LIN {X 0,Y 369.377,Z 414.803,A -85,B 0,C 180,E1 -12869.73,E2 -12869.73} C_VEL
LIN {X 0,Y 368.676,Z 422.155,A -85,B 0,C 180,E1 -12871.367,E2 -12871.367} C_VEL
LIN {X 0,Y 368.229,Z 428.905,A -85,B 0,C 180,E1 -12873.284,E2 -12873.284} C_VEL
LIN {X 0,Y 367.894,Z 433.372,A -85,B 0,C 180,E1 -12874.933,E2 -12874.933} C_VEL
LIN {X 0,Y 367.73,Z 436.765,A -85,B 0,C 180,E1 -12876.586,E2 -12876.586} C_VEL
LIN {X 0,Y 367.581,Z 438.459,A -85,B 0,C 180,E1 -12877.693,E2 -12877.693} C_VEL
LIN {X 0,Y 367.47,Z 439.751,A -85,B 0,C 180,E1 -12878.802,E2 -12878.802} C_VEL
LIN {X 0,Y 367.38,Z 440.649,A -85,B 0,C 180,E1 -12879.915,E2 -12879.915} C_VEL
LIN {X 0,Y 367.424,Z 441.1,A -85,B 0,C 180,E1 -12881.028,E2 -12881.028} C_VEL
LIN {X 0,Y 367.521,Z 441.023,A -85,B 0,C 180,E1 -12882.77,E2 -12882.77} C_VEL
LIN {X 0,Y 367.587,Z 440.078,A -85,B 0,C 180,E1 -12884.392,E2 -12884.392} C_VEL
LIN {X 0,Y 367.854,Z 438.002,A -85,B 0,C 180,E1 -12886.13,E2 -12886.13} C_VEL
LIN {X 0,Y 368.254,Z 435.208,A -85,B 0,C 180,E1 -12887.78,E2 -12887.78} C_VEL
LIN {X 0,Y 368.738,Z 431.176,A -85,B 0,C 180,E1 -12889.484,E2 -12889.484} C_VEL
LIN {X 0,Y 369.195,Z 427.833,A -85,B 0,C 180,E1 -12890.605,E2 -12890.605} C_VEL
LIN {X 0,Y 368.924,Z 425.231,A -85,B 0,C 180,E1 -12891.428,E2 -12891.428} C_VEL
LIN {X 0,Y 366.799,Z 420.655,A -85,B 0,C 180,E1 -12892.758,E2 -12892.758} C_VEL
LIN {X 0,Y 364.754,Z 415.467,A -85,B 0,C 180,E1 -12894.041,E2 -12894.041} C_VEL
LIN {X 0,Y 364.604,Z 411.868,A -85,B 0,C 180,E1 -12894.779,E2 -12894.779} C_VEL
LIN {X 0,Y 365.717,Z 403.299,A -85,B 0,C 180,E1 -12896.231,E2 -12896.231} C_VEL
LIN {X 0,Y 366.895,Z 393.904,A -85,B 0,C 180,E1 -12897.523,E2 -12897.523} C_VEL
LIN {X 0,Y 368.133,Z 383.723,A -85,B 0,C 180,E1 -12898.647,E2 -12898.647} C_VEL
LIN {X 0,Y 369.203,Z 372.197,A -85,B 0,C 180,E1 -12899.664,E2 -12899.664} C_VEL
LIN {X 0,Y 370.055,Z 360.622,A -85,B 0,C 180,E1 -12900.453,E2 -12900.453} C_VEL
LIN {X 0,Y 370.819,Z 347.971,A -85,B 0,C 180,E1 -12901.072,E2 -12901.072} C_VEL
LIN {X 0,Y 371.327,Z 334.426,A -85,B 0,C 180,E1 -12901.491,E2 -12901.491} C_VEL
LIN {X 0,Y 372.84,Z 255.873,A -85,B 0,C 180,E1 -12903.038,E2 -12903.038} C_VEL
LIN {X 0,Y 370.773,Z 248.12,A -85,B 0,C 180,E1 -12903.357,E2 -12903.357} C_VEL
LIN {X 0,Y 363.463,Z 231.06,A -85,B 0,C 180,E1 -12904.307,E2 -12904.307} C_VEL
LIN {X 0,Y 361.887,Z 224.41,A -85,B 0,C 180,E1 -12906.234,E2 -12906.234} C_VEL
LIN {X 0,Y 361.876,Z 224.407,A -85,B 0,C 180,E1 -12909.857,E2 -12909.857} C_VEL
LIN {X 0,Y 361.848,Z 224.414,A -85,B 0,C 180,E1 -12912.825,E2 -12912.825} C_VEL
LIN {X 0,Y 361.888,Z 224.41,A -85,B 0,C 180,E1 -12915.932,E2 -12915.932} C_VEL
LIN {X 0,Y 361.896,Z 224.406,A -85,B 0,C 180,E1 -12919.23,E2 -12919.23} C_VEL
LIN {X 0,Y 361.856,Z 224.406,A -85,B 0,C 180,E1 -12922.98,E2 -12922.98} C_VEL
LIN {X 0,Y 361.845,Z 224.411,A -85,B 0,C 180,E1 -12926.629,E2 -12926.629} C_VEL
LIN {X 0,Y 361.861,Z 224.406,A -85,B 0,C 180,E1 -12929.67,E2 -12929.67} C_VEL
LIN {X 0,Y 361.937,Z 224.396,A -85,B 0,C 180,E1 -12933.473,E2 -12933.473} C_VEL
LIN {X 0,Y 361.859,Z 224.404,A -85,B 0,C 180,E1 -12937.142,E2 -12937.142} C_VEL
LIN {X 0,Y 361.862,Z 224.401,A -85,B 0,C 180,E1 -12940.721,E2 -12940.721} C_VEL
LIN {X 0,Y 361.912,Z 224.403,A -85,B 0,C 180,E1 -12943.065,E2 -12943.065} C_VEL
LIN {X 0,Y 361.976,Z 224.393,A -85,B 0,C 180,E1 -12946.527,E2 -12946.527} C_VEL
LIN {X 0,Y 362.007,Z 224.39,A -85,B 0,C 180,E1 -12949.937,E2 -12949.937} C_VEL
LIN {X 0,Y 362.141,Z 224.37,A -85,B 0,C 180,E1 -12953.313,E2 -12953.313} C_VEL
LIN {X 0,Y 362.252,Z 224.352,A -85,B 0,C 180,E1 -12957.776,E2 -12957.776} C_VEL
LIN {X 0,Y 362.379,Z 224.343,A -85,B 0,C 180,E1 -12960,E2 -12960} C_VEL
LIN {X 0,Y 362.252,Z 224.355,A -85,B 0,C 180,E1 -12962.224,E2 -12962.224} C_VEL
LIN {X 0,Y 362.113,Z 224.377,A -85,B 0,C 180,E1 -12966.687,E2 -12966.687} C_VEL
LIN {X 0,Y 361.977,Z 224.393,A -85,B 0,C 180,E1 -12970.063,E2 -12970.063} C_VEL
LIN {X 0,Y 361.977,Z 224.392,A -85,B 0,C 180,E1 -12973.899,E2 -12973.899} C_VEL
LIN {X 0,Y 361.907,Z 224.398,A -85,B 0,C 180,E1 -12976.935,E2 -12976.935} C_VEL
LIN {X 0,Y 361.854,Z 224.409,A -85,B 0,C 180,E1 -12980.463,E2 -12980.463} C_VEL
LIN {X 0,Y 361.843,Z 224.411,A -85,B 0,C 180,E1 -12984.102,E2 -12984.102} C_VEL
LIN {X 0,Y 361.826,Z 224.413,A -85,B 0,C 180,E1 -12987.786,E2 -12987.786} C_VEL
LIN {X 0,Y 361.81,Z 224.415,A -85,B 0,C 180,E1 -12991.281,E2 -12991.281} C_VEL
LIN {X 0,Y 361.835,Z 224.408,A -85,B 0,C 180,E1 -12994.283,E2 -12994.283} C_VEL
LIN {X 0,Y 361.845,Z 224.4,A -85,B 0,C 180,E1 -12997.223,E2 -12997.223} C_VEL
LIN {X 0,Y 361.822,Z 224.415,A -85,B 0,C 180,E1 -13000.756,E2 -13000.756} C_VEL
LIN {X 0,Y 361.806,Z 224.418,A -85,B 0,C 180,E1 -13004.37,E2 -13004.37} C_VEL
LIN {X 0,Y 361.822,Z 224.41,A -85,B 0,C 180,E1 -13007.571,E2 -13007.571} C_VEL
LIN {X 0,Y 361.836,Z 224.407,A -85,B 0,C 180,E1 -13011.573,E2 -13011.573} C_VEL
LIN {X 0,Y 361.87,Z 224.404,A -85,B 0,C 180,E1 -13014.656,E2 -13014.656} C_VEL
LIN {X 0,Y 361.907,Z 224.589,A -85,B 0,C 180,E1 -13018.051,E2 -13018.051} C_VEL
LIN {X 0,Y 365.046,Z 237.635,A -85,B 0,C 180,E1 -13021.507,E2 -13021.507} C_VEL
LIN {X 0,Y 366.873,Z 247.039,A -85,B 0,C 180,E1 -13023.858,E2 -13023.858} C_VEL
LIN {X 0,Y 366,Z 256.31,A -85,B 0,C 180,E1 -13025.918,E2 -13025.918} C_VEL
LIN {X 0,Y 365.489,Z 261.029,A -85,B 0,C 180,E1 -13026.928,E2 -13026.928} C_VEL
LIN {X 0,Y 370.101,Z 284.638,A -85,B 0,C 180,E1 -13027.78,E2 -13027.78} C_VEL
LIN {X 0,Y 372.121,Z 298.577,A -85,B 0,C 180,E1 -13028.219,E2 -13028.219} C_VEL
LIN {X 0,Y 370.713,Z 370.18,A -85,B 0,C 180,E1 -13029.649,E2 -13029.649} C_VEL
LIN {X 0,Y 369.936,Z 383.988,A -85,B 0,C 180,E1 -13030.148,E2 -13030.148} C_VEL
LIN {X 0,Y 368.872,Z 396.399,A -85,B 0,C 180,E1 -13030.812,E2 -13030.812} C_VEL
LIN {X 0,Y 367.758,Z 407.492,A -85,B 0,C 180,E1 -13031.619,E2 -13031.619} C_VEL
LIN {X 0,Y 366.392,Z 419.049,A -85,B 0,C 180,E1 -13032.703,E2 -13032.703} C_VEL
LIN {X 0,Y 365.116,Z 429.47,A -85,B 0,C 180,E1 -13033.936,E2 -13033.936} C_VEL
LIN {X 0,Y 363.969,Z 438.334,A -85,B 0,C 180,E1 -13035.227,E2 -13035.227} C_VEL
LIN {X 0,Y 362.841,Z 447.307,A -85,B 0,C 180,E1 -13036.844,E2 -13036.844} C_VEL
LIN {X 0,Y 361.793,Z 454.782,A -85,B 0,C 180,E1 -13038.514,E2 -13038.514} C_VEL
LIN {X 0,Y 361.043,Z 461.718,A -85,B 0,C 180,E1 -13040.475,E2 -13040.475} C_VEL
LIN {X 0,Y 360.649,Z 466.318,A -85,B 0,C 180,E1 -13042.159,E2 -13042.159} C_VEL
LIN {X 0,Y 360.424,Z 470.058,A -85,B 0,C 180,E1 -13043.969,E2 -13043.969} C_VEL
LIN {X 0,Y 360.364,Z 472.357,A -85,B 0,C 180,E1 -13045.524,E2 -13045.524} C_VEL
LIN {X 0,Y 360.321,Z 473.53,A -85,B 0,C 180,E1 -13046.644,E2 -13046.644} C_VEL
LIN {X 0,Y 360.454,Z 474.635,A -85,B 0,C 180,E1 -13048.881,E2 -13048.881} C_VEL
LIN {X 0,Y 360.48,Z 474.606,A -85,B 0,C 180,E1 -13049.998,E2 -13049.998} C_VEL
LIN {X 0,Y 360.476,Z 474.176,A -85,B 0,C 180,E1 -13051.115,E2 -13051.115} C_VEL
LIN {X 0,Y 360.395,Z 473.302,A -85,B 0,C 180,E1 -13052.233,E2 -13052.233} C_VEL
LIN {X 0,Y 360.436,Z 470.349,A -85,B 0,C 180,E1 -13054.471,E2 -13054.471} C_VEL
LIN {X 0,Y 360.442,Z 467.158,A -85,B 0,C 180,E1 -13056.059,E2 -13056.059} C_VEL
LIN {X 0,Y 360.637,Z 462.452,A -85,B 0,C 180,E1 -13057.837,E2 -13057.837} C_VEL
LIN {X 0,Y 361.013,Z 455.625,A -85,B 0,C 180,E1 -13059.804,E2 -13059.804} C_VEL
LIN {X 0,Y 361.56,Z 448.175,A -85,B 0,C 180,E1 -13061.489,E2 -13061.489} C_VEL
LIN {X 0,Y 362.248,Z 440.586,A -85,B 0,C 180,E1 -13062.888,E2 -13062.888} C_VEL
LIN {X 0,Y 363.021,Z 432.028,A -85,B 0,C 180,E1 -13064.194,E2 -13064.194} C_VEL
LIN {X 0,Y 363.918,Z 421.306,A -85,B 0,C 180,E1 -13065.524,E2 -13065.524} C_VEL
LIN {X 0,Y 364.862,Z 409.823,A -85,B 0,C 180,E1 -13066.646,E2 -13066.646} C_VEL
LIN {X 0,Y 365.769,Z 398.067,A -85,B 0,C 180,E1 -13067.539,E2 -13067.539} C_VEL
LIN {X 0,Y 366.614,Z 385.299,A -85,B 0,C 180,E1 -13068.255,E2 -13068.255} C_VEL
LIN {X 0,Y 367.305,Z 371.702,A -85,B 0,C 180,E1 -13068.761,E2 -13068.761} C_VEL
LIN {X 0,Y 367.865,Z 337.148,A -85,B 0,C 180,E1 -13069.469,E2 -13069.469} C_VEL
LIN {X 0,Y 368.221,Z 295.328,A -85,B 0,C 180,E1 -13070.291,E2 -13070.291} C_VEL
LIN {X 0,Y 363.689,Z 261.477,A -85,B 0,C 180,E1 -13071.21,E2 -13071.21} C_VEL
LIN {X 0,Y 365.131,Z 243.552,A -85,B 0,C 180,E1 -13075.048,E2 -13075.048} C_VEL
LIN {X 0,Y 364.937,Z 239.311,A -85,B 0,C 180,E1 -13075.993,E2 -13075.993} C_VEL
LIN {X 0,Y 362.387,Z 226.582,A -85,B 0,C 180,E1 -13078.997,E2 -13078.997} C_VEL
LIN {X 0,Y 361.891,Z 224.407,A -85,B 0,C 180,E1 -13079.546,E2 -13079.546} C_VEL
LIN {X 0,Y 361.841,Z 224.41,A -85,B 0,C 180,E1 -13083.365,E2 -13083.365} C_VEL
LIN {X 0,Y 361.846,Z 224.408,A -85,B 0,C 180,E1 -13087.014,E2 -13087.014} C_VEL
LIN {X 0,Y 361.831,Z 224.416,A -85,B 0,C 180,E1 -13089.857,E2 -13089.857} C_VEL
LIN {X 0,Y 361.812,Z 224.413,A -85,B 0,C 180,E1 -13092.824,E2 -13092.824} C_VEL
LIN {X 0,Y 361.868,Z 224.411,A -85,B 0,C 180,E1 -13095.93,E2 -13095.93} C_VEL
LIN {X 0,Y 361.876,Z 224.406,A -85,B 0,C 180,E1 -13099.228,E2 -13099.228} C_VEL
LIN {X 0,Y 361.834,Z 224.41,A -85,B 0,C 180,E1 -13102.978,E2 -13102.978} C_VEL
LIN {X 0,Y 361.822,Z 224.411,A -85,B 0,C 180,E1 -13106.627,E2 -13106.627} C_VEL
LIN {X 0,Y 361.837,Z 224.415,A -85,B 0,C 180,E1 -13109.669,E2 -13109.669} C_VEL
LIN {X 0,Y 361.913,Z 224.406,A -85,B 0,C 180,E1 -13113.472,E2 -13113.472} C_VEL
LIN {X 0,Y 361.879,Z 224.407,A -85,B 0,C 180,E1 -13117.144,E2 -13117.144} C_VEL
LIN {X 0,Y 361.89,Z 224.404,A -85,B 0,C 180,E1 -13120.722,E2 -13120.722} C_VEL
LIN {X 0,Y 361.9,Z 224.402,A -85,B 0,C 180,E1 -13124.224,E2 -13124.224} C_VEL
LIN {X 0,Y 361.952,Z 224.395,A -85,B 0,C 180,E1 -13126.526,E2 -13126.526} C_VEL
LIN {X 0,Y 361.988,Z 224.391,A -85,B 0,C 180,E1 -13129.937,E2 -13129.937} C_VEL
LIN {X 0,Y 362.101,Z 224.377,A -85,B 0,C 180,E1 -13132.192,E2 -13132.192} C_VEL
LIN {X 0,Y 362.075,Z 224.38,A -85,B 0,C 180,E1 -13134.431,E2 -13134.431} C_VEL
LIN {X 0,Y 362.232,Z 224.361,A -85,B 0,C 180,E1 -13137.776,E2 -13137.776} C_VEL
LIN {X 0,Y 362.376,Z 224.342,A -85,B 0,C 180,E1 -13140,E2 -13140} C_VEL
LIN {X 0,Y 362.228,Z 224.361,A -85,B 0,C 180,E1 -13142.224,E2 -13142.224} C_VEL
LIN {X 0,Y 362.111,Z 224.379,A -85,B 0,C 180,E1 -13146.687,E2 -13146.687} C_VEL
LIN {X 0,Y 361.985,Z 224.391,A -85,B 0,C 180,E1 -13150.063,E2 -13150.063} C_VEL
LIN {X 0,Y 361.952,Z 224.395,A -85,B 0,C 180,E1 -13153.9,E2 -13153.9} C_VEL
LIN {X 0,Y 361.908,Z 224.401,A -85,B 0,C 180,E1 -13157.933,E2 -13157.933} C_VEL
LIN {X 0,Y 361.817,Z 224.412,A -85,B 0,C 180,E1 -13161.658,E2 -13161.658} C_VEL
LIN {X 0,Y 361.884,Z 224.404,A -85,B 0,C 180,E1 -13165.294,E2 -13165.294} C_VEL
LIN {X 0,Y 361.879,Z 224.405,A -85,B 0,C 180,E1 -13167.782,E2 -13167.782} C_VEL
LIN {X 0,Y 361.81,Z 224.413,A -85,B 0,C 180,E1 -13171.289,E2 -13171.289} C_VEL
LIN {X 0,Y 361.818,Z 224.416,A -85,B 0,C 180,E1 -13174.285,E2 -13174.285} C_VEL
LIN {X 0,Y 361.83,Z 224.41,A -85,B 0,C 180,E1 -13177.227,E2 -13177.227} C_VEL
LIN {X 0,Y 361.877,Z 224.407,A -85,B 0,C 180,E1 -13180.773,E2 -13180.773} C_VEL
LIN {X 0,Y 361.874,Z 224.41,A -85,B 0,C 180,E1 -13184.36,E2 -13184.36} C_VEL
LIN {X 0,Y 361.812,Z 224.413,A -85,B 0,C 180,E1 -13187.573,E2 -13187.573} C_VEL
LIN {X 0,Y 361.848,Z 224.408,A -85,B 0,C 180,E1 -13190.978,E2 -13190.978} C_VEL
LIN {X 0,Y 361.856,Z 224.408,A -85,B 0,C 180,E1 -13194.66,E2 -13194.66} C_VEL
LIN {X 0,Y 361.823,Z 224.414,A -85,B 0,C 180,E1 -13198.375,E2 -13198.375} C_VEL
LIN {X 0,Y 361.896,Z 224.406,A -85,B 0,C 180,E1 -13202.225,E2 -13202.225} C_VEL
LIN {X 0,Y 361.917,Z 224.4,A -85,B 0,C 180,E1 -13204.714,E2 -13204.714} C_VEL
LIN {X 0,Y 361.854,Z 224.409,A -85,B 0,C 180,E1 -13208.349,E2 -13208.349} C_VEL
LIN {X 0,Y 361.916,Z 224.403,A -85,B 0,C 180,E1 -13212.088,E2 -13212.088} C_VEL
LIN {X 0,Y 361.959,Z 224.397,A -85,B 0,C 180,E1 -13215.383,E2 -13215.383} C_VEL
LIN {X 0,Y 362.005,Z 224.579,A -85,B 0,C 180,E1 -13218.312,E2 -13218.312} C_VEL
LIN {X 0,Y 363.238,Z 230.767,A -85,B 0,C 180,E1 -13219.872,E2 -13219.872} C_VEL
LIN {X 0,Y 366.475,Z 241.241,A -85,B 0,C 180,E1 -13220.25,E2 -13220.25} C_VEL
LIN {X 0,Y 368.895,Z 254.352,A -85,B 0,C 180,E1 -13220.635,E2 -13220.635} C_VEL
LIN {X 0,Y 367.507,Z 337.938,A -85,B 0,C 180,E1 -13222.275,E2 -13222.275} C_VEL
LIN {X 0,Y 367.022,Z 351.062,A -85,B 0,C 180,E1 -13222.749,E2 -13222.749} C_VEL
LIN {X 0,Y 366.477,Z 363.096,A -85,B 0,C 180,E1 -13223.395,E2 -13223.395} C_VEL
LIN {X 0,Y 365.943,Z 374.427,A -85,B 0,C 180,E1 -13224.216,E2 -13224.216} C_VEL
LIN {X 0,Y 364.895,Z 386.165,A -85,B 0,C 180,E1 -13225.307,E2 -13225.307} C_VEL
LIN {X 0,Y 364.001,Z 396.644,A -85,B 0,C 180,E1 -13226.543,E2 -13226.543} C_VEL
LIN {X 0,Y 363.227,Z 405.215,A -85,B 0,C 180,E1 -13227.785,E2 -13227.785} C_VEL
LIN {X 0,Y 362.557,Z 413.108,A -85,B 0,C 180,E1 -13229.169,E2 -13229.169} C_VEL
LIN {X 0,Y 361.754,Z 420.868,A -85,B 0,C 180,E1 -13230.837,E2 -13230.837} C_VEL
LIN {X 0,Y 361.263,Z 427.957,A -85,B 0,C 180,E1 -13232.789,E2 -13232.789} C_VEL
LIN {X 0,Y 360.853,Z 432.71,A -85,B 0,C 180,E1 -13234.47,E2 -13234.47} C_VEL
LIN {X 0,Y 360.675,Z 436.807,A -85,B 0,C 180,E1 -13236.396,E2 -13236.396} C_VEL
LIN {X 0,Y 360.469,Z 438.987,A -85,B 0,C 180,E1 -13237.845,E2 -13237.845} C_VEL
LIN {X 0,Y 360.38,Z 440.234,A -85,B 0,C 180,E1 -13238.977,E2 -13238.977} C_VEL
LIN {X 0,Y 360.286,Z 441.057,A -85,B 0,C 180,E1 -13240.112,E2 -13240.112} C_VEL
LIN {X 0,Y 360.358,Z 441.451,A -85,B 0,C 180,E1 -13241.247,E2 -13241.247} C_VEL
LIN {X 0,Y 360.451,Z 441.352,A -85,B 0,C 180,E1 -13242.865,E2 -13242.865} C_VEL
LIN {X 0,Y 360.539,Z 440.257,A -85,B 0,C 180,E1 -13244.68,E2 -13244.68} C_VEL
LIN {X 0,Y 360.713,Z 439.007,A -85,B 0,C 180,E1 -13245.83,E2 -13245.83} C_VEL
LIN {X 0,Y 361.123,Z 436.391,A -85,B 0,C 180,E1 -13247.519,E2 -13247.519} C_VEL
LIN {X 0,Y 361.609,Z 432.561,A -85,B 0,C 180,E1 -13249.293,E2 -13249.293} C_VEL
LIN {X 0,Y 362.309,Z 427.786,A -85,B 0,C 180,E1 -13250.974,E2 -13250.974} C_VEL
LIN {X 0,Y 363.2,Z 421.309,A -85,B 0,C 180,E1 -13252.768,E2 -13252.768} C_VEL
LIN {X 0,Y 364.407,Z 413.357,A -85,B 0,C 180,E1 -13254.497,E2 -13254.497} C_VEL
LIN {X 0,Y 364.604,Z 411.868,A -85,B 0,C 180,E1 -13254.779,E2 -13254.779} C_VEL
LIN {X 0,Y 364.459,Z 408.101,A -85,B 0,C 180,E1 -13255.497,E2 -13255.497} C_VEL
LIN {X 0,Y 362.508,Z 401.791,A -85,B 0,C 180,E1 -13256.667,E2 -13256.667} C_VEL
LIN {X 0,Y 360.686,Z 395.024,A -85,B 0,C 180,E1 -13257.77,E2 -13257.77} C_VEL
LIN {X 0,Y 360.713,Z 390.444,A -85,B 0,C 180,E1 -13258.363,E2 -13258.363} C_VEL
LIN {X 0,Y 362.021,Z 379.271,A -85,B 0,C 180,E1 -13259.512,E2 -13259.512} C_VEL
LIN {X 0,Y 363.107,Z 366.471,A -85,B 0,C 180,E1 -13260.535,E2 -13260.535} C_VEL
LIN {X 0,Y 364.007,Z 354.12,A -85,B 0,C 180,E1 -13261.256,E2 -13261.256} C_VEL
LIN {X 0,Y 364.648,Z 340.948,A -85,B 0,C 180,E1 -13261.777,E2 -13261.777} C_VEL
LIN {X 0,Y 365.172,Z 319.833,A -85,B 0,C 180,E1 -13262.245,E2 -13262.245} C_VEL
LIN {X 0,Y 366.417,Z 257.084,A -85,B 0,C 180,E1 -13263.497,E2 -13263.497} C_VEL
LIN {X 0,Y 364.527,Z 250.334,A -85,B 0,C 180,E1 -13263.791,E2 -13263.791} C_VEL
LIN {X 0,Y 356.336,Z 231.44,A -85,B 0,C 180,E1 -13264.886,E2 -13264.886} C_VEL
LIN {X 0,Y 354.841,Z 225.287,A -85,B 0,C 180,E1 -13266.718,E2 -13266.718} C_VEL
LIN {X 0,Y 354.82,Z 225.289,A -85,B 0,C 180,E1 -13269.422,E2 -13269.422} C_VEL
LIN {X 0,Y 354.8,Z 225.292,A -85,B 0,C 180,E1 -13272.869,E2 -13272.869} C_VEL
LIN {X 0,Y 354.831,Z 225.291,A -85,B 0,C 180,E1 -13276.113,E2 -13276.113} C_VEL
LIN {X 0,Y 354.847,Z 225.284,A -85,B 0,C 180,E1 -13279.187,E2 -13279.187} C_VEL
LIN {X 0,Y 354.797,Z 225.286,A -85,B 0,C 180,E1 -13282.401,E2 -13282.401} C_VEL
LIN {X 0,Y 354.799,Z 225.287,A -85,B 0,C 180,E1 -13284.939,E2 -13284.939} C_VEL
LIN {X 0,Y 354.779,Z 225.287,A -85,B 0,C 180,E1 -13288.404,E2 -13288.404} C_VEL
LIN {X 0,Y 354.836,Z 225.284,A -85,B 0,C 180,E1 -13291.617,E2 -13291.617} C_VEL
LIN {X 0,Y 354.881,Z 225.28,A -85,B 0,C 180,E1 -13294.171,E2 -13294.171} C_VEL
LIN {X 0,Y 354.796,Z 225.292,A -85,B 0,C 180,E1 -13297.891,E2 -13297.891} C_VEL
LIN {X 0,Y 354.904,Z 225.278,A -85,B 0,C 180,E1 -13301.891,E2 -13301.891} C_VEL
LIN {X 0,Y 354.922,Z 225.274,A -85,B 0,C 180,E1 -13305.982,E2 -13305.982} C_VEL
LIN {X 0,Y 354.954,Z 225.267,A -85,B 0,C 180,E1 -13309.735,E2 -13309.735} C_VEL
LIN {X 0,Y 355.104,Z 225.247,A -85,B 0,C 180,E1 -13313.18,E2 -13313.18} C_VEL
LIN {X 0,Y 355.216,Z 225.229,A -85,B 0,C 180,E1 -13317.732,E2 -13317.732} C_VEL
LIN {X 0,Y 355.329,Z 225.221,A -85,B 0,C 180,E1 -13320,E2 -13320} C_VEL
LIN {X 0,Y 355.215,Z 225.232,A -85,B 0,C 180,E1 -13322.268,E2 -13322.268} C_VEL
LIN {X 0,Y 355.077,Z 225.251,A -85,B 0,C 180,E1 -13326.82,E2 -13326.82} C_VEL
LIN {X 0,Y 354.934,Z 225.27,A -85,B 0,C 180,E1 -13330.265,E2 -13330.265} C_VEL
LIN {X 0,Y 354.921,Z 225.271,A -85,B 0,C 180,E1 -13334.018,E2 -13334.018} C_VEL
LIN {X 0,Y 354.869,Z 225.275,A -85,B 0,C 180,E1 -13338.092,E2 -13338.092} C_VEL
LIN {X 0,Y 354.787,Z 225.283,A -85,B 0,C 180,E1 -13342.109,E2 -13342.109} C_VEL
LIN {X 0,Y 354.789,Z 225.281,A -85,B 0,C 180,E1 -13345.836,E2 -13345.836} C_VEL
LIN {X 0,Y 354.777,Z 225.285,A -85,B 0,C 180,E1 -13349.686,E2 -13349.686} C_VEL
LIN {X 0,Y 354.793,Z 225.282,A -85,B 0,C 180,E1 -13353.703,E2 -13353.703} C_VEL
LIN {X 0,Y 354.779,Z 225.286,A -85,B 0,C 180,E1 -13356.462,E2 -13356.462} C_VEL
LIN {X 0,Y 354.788,Z 225.275,A -85,B 0,C 180,E1 -13359.42,E2 -13359.42} C_VEL
LIN {X 0,Y 354.777,Z 225.29,A -85,B 0,C 180,E1 -13362.868,E2 -13362.868} C_VEL
LIN {X 0,Y 354.757,Z 225.296,A -85,B 0,C 180,E1 -13366.105,E2 -13366.105} C_VEL
LIN {X 0,Y 354.759,Z 225.29,A -85,B 0,C 180,E1 -13369.177,E2 -13369.177} C_VEL
LIN {X 0,Y 354.795,Z 225.286,A -85,B 0,C 180,E1 -13372.405,E2 -13372.405} C_VEL
LIN {X 0,Y 354.808,Z 225.284,A -85,B 0,C 180,E1 -13374.942,E2 -13374.942} C_VEL
LIN {X 0,Y 354.829,Z 225.45,A -85,B 0,C 180,E1 -13377.546,E2 -13377.546} C_VEL
LIN {X 0,Y 358.154,Z 239.13,A -85,B 0,C 180,E1 -13381.266,E2 -13381.266} C_VEL
LIN {X 0,Y 360.021,Z 248.666,A -85,B 0,C 180,E1 -13383.703,E2 -13383.703} C_VEL
LIN {X 0,Y 359.01,Z 258.823,A -85,B 0,C 180,E1 -13386.003,E2 -13386.003} C_VEL
LIN {X 0,Y 358.787,Z 260.543,A -85,B 0,C 180,E1 -13386.386,E2 -13386.386} C_VEL
LIN {X 0,Y 363.779,Z 286.169,A -85,B 0,C 180,E1 -13387.34,E2 -13387.34} C_VEL
LIN {X 0,Y 365.668,Z 298.645,A -85,B 0,C 180,E1 -13387.75,E2 -13387.75} C_VEL
LIN {X 0,Y 364.246,Z 369.797,A -85,B 0,C 180,E1 -13389.198,E2 -13389.198} C_VEL
LIN {X 0,Y 363.407,Z 383.627,A -85,B 0,C 180,E1 -13389.702,E2 -13389.702} C_VEL
LIN {X 0,Y 362.335,Z 396.043,A -85,B 0,C 180,E1 -13390.379,E2 -13390.379} C_VEL
LIN {X 0,Y 361.057,Z 407.925,A -85,B 0,C 180,E1 -13391.266,E2 -13391.266} C_VEL
LIN {X 0,Y 359.615,Z 419.337,A -85,B 0,C 180,E1 -13392.367,E2 -13392.367} C_VEL
LIN {X 0,Y 358.293,Z 429.646,A -85,B 0,C 180,E1 -13393.622,E2 -13393.622} C_VEL
LIN {X 0,Y 357.054,Z 438.701,A -85,B 0,C 180,E1 -13394.985,E2 -13394.985} C_VEL
LIN {X 0,Y 355.922,Z 447.287,A -85,B 0,C 180,E1 -13396.583,E2 -13396.583} C_VEL
LIN {X 0,Y 354.824,Z 454.708,A -85,B 0,C 180,E1 -13398.285,E2 -13398.285} C_VEL
LIN {X 0,Y 354.013,Z 461.581,A -85,B 0,C 180,E1 -13400.284,E2 -13400.284} C_VEL
LIN {X 0,Y 353.576,Z 466.136,A -85,B 0,C 180,E1 -13402.001,E2 -13402.001} C_VEL
LIN {X 0,Y 353.317,Z 470.12,A -85,B 0,C 180,E1 -13404.03,E2 -13404.03} C_VEL
LIN {X 0,Y 353.277,Z 472.111,A -85,B 0,C 180,E1 -13405.434,E2 -13405.434} C_VEL
LIN {X 0,Y 353.241,Z 473.248,A -85,B 0,C 180,E1 -13406.576,E2 -13406.576} C_VEL
LIN {X 0,Y 353.356,Z 474.316,A -85,B 0,C 180,E1 -13408.858,E2 -13408.858} C_VEL
LIN {X 0,Y 353.398,Z 474.27,A -85,B 0,C 180,E1 -13409.998,E2 -13409.998} C_VEL
LIN {X 0,Y 353.394,Z 473.806,A -85,B 0,C 180,E1 -13411.137,E2 -13411.137} C_VEL
LIN {X 0,Y 353.271,Z 471.617,A -85,B 0,C 180,E1 -13413.419,E2 -13413.419} C_VEL
LIN {X 0,Y 353.319,Z 468.866,A -85,B 0,C 180,E1 -13415.133,E2 -13415.133} C_VEL
LIN {X 0,Y 353.414,Z 465.071,A -85,B 0,C 180,E1 -13416.85,E2 -13416.85} C_VEL
LIN {X 0,Y 353.644,Z 460.134,A -85,B 0,C 180,E1 -13418.569,E2 -13418.569} C_VEL
LIN {X 0,Y 354.035,Z 453.903,A -85,B 0,C 180,E1 -13420.289,E2 -13420.289} C_VEL
LIN {X 0,Y 354.724,Z 446.142,A -85,B 0,C 180,E1 -13422.004,E2 -13422.004} C_VEL
LIN {X 0,Y 355.621,Z 436.374,A -85,B 0,C 180,E1 -13423.715,E2 -13423.715} C_VEL
LIN {X 0,Y 356.322,Z 428.247,A -85,B 0,C 180,E1 -13424.88,E2 -13424.88} C_VEL
LIN {X 0,Y 357.264,Z 417.633,A -85,B 0,C 180,E1 -13426.129,E2 -13426.129} C_VEL
LIN {X 0,Y 358.189,Z 407.161,A -85,B 0,C 180,E1 -13427.112,E2 -13427.112} C_VEL
LIN {X 0,Y 359.125,Z 394.557,A -85,B 0,C 180,E1 -13428.022,E2 -13428.022} C_VEL
LIN {X 0,Y 360.012,Z 381.267,A -85,B 0,C 180,E1 -13428.712,E2 -13428.712} C_VEL
LIN {X 0,Y 360.514,Z 369.174,A -85,B 0,C 180,E1 -13429.128,E2 -13429.128} C_VEL
LIN {X 0,Y 361.556,Z 297.335,A -85,B 0,C 180,E1 -13430.567,E2 -13430.567} C_VEL
LIN {X 0,Y 356.752,Z 261.183,A -85,B 0,C 180,E1 -13431.561,E2 -13431.561} C_VEL
LIN {X 0,Y 358.058,Z 245.629,A -85,B 0,C 180,E1 -13434.956,E2 -13434.956} C_VEL
LIN {X 0,Y 358.114,Z 241.476,A -85,B 0,C 180,E1 -13435.886,E2 -13435.886} C_VEL
LIN {X 0,Y 355.615,Z 228.716,A -85,B 0,C 180,E1 -13438.946,E2 -13438.946} C_VEL
LIN {X 0,Y 354.837,Z 225.286,A -85,B 0,C 180,E1 -13439.838,E2 -13439.838} C_VEL
LIN {X 0,Y 354.789,Z 225.29,A -85,B 0,C 180,E1 -13443.698,E2 -13443.698} C_VEL
LIN {X 0,Y 354.777,Z 225.291,A -85,B 0,C 180,E1 -13446.455,E2 -13446.455} C_VEL
LIN {X 0,Y 354.802,Z 225.287,A -85,B 0,C 180,E1 -13449.419,E2 -13449.419} C_VEL
LIN {X 0,Y 354.764,Z 225.291,A -85,B 0,C 180,E1 -13452.863,E2 -13452.863} C_VEL
LIN {X 0,Y 354.811,Z 225.288,A -85,B 0,C 180,E1 -13456.11,E2 -13456.11} C_VEL
LIN {X 0,Y 354.827,Z 225.284,A -85,B 0,C 180,E1 -13459.184,E2 -13459.184} C_VEL
LIN {X 0,Y 354.775,Z 225.29,A -85,B 0,C 180,E1 -13462.398,E2 -13462.398} C_VEL
LIN {X 0,Y 354.776,Z 225.29,A -85,B 0,C 180,E1 -13464.937,E2 -13464.937} C_VEL
LIN {X 0,Y 354.755,Z 225.292,A -85,B 0,C 180,E1 -13468.402,E2 -13468.402} C_VEL
LIN {X 0,Y 354.812,Z 225.29,A -85,B 0,C 180,E1 -13471.616,E2 -13471.616} C_VEL
LIN {X 0,Y 354.859,Z 225.279,A -85,B 0,C 180,E1 -13474.169,E2 -13474.169} C_VEL
LIN {X 0,Y 354.849,Z 225.282,A -85,B 0,C 180,E1 -13477.895,E2 -13477.895} C_VEL
LIN {X 0,Y 354.879,Z 225.278,A -85,B 0,C 180,E1 -13481.889,E2 -13481.889} C_VEL
LIN {X 0,Y 354.896,Z 225.275,A -85,B 0,C 180,E1 -13485.98,E2 -13485.98} C_VEL
LIN {X 0,Y 354.935,Z 225.271,A -85,B 0,C 180,E1 -13489.735,E2 -13489.735} C_VEL
LIN {X 0,Y 355.082,Z 225.251,A -85,B 0,C 180,E1 -13492.036,E2 -13492.036} C_VEL
LIN {X 0,Y 355.049,Z 225.255,A -85,B 0,C 180,E1 -13494.32,E2 -13494.32} C_VEL
LIN {X 0,Y 355.196,Z 225.238,A -85,B 0,C 180,E1 -13497.732,E2 -13497.732} C_VEL
LIN {X 0,Y 355.325,Z 225.221,A -85,B 0,C 180,E1 -13500,E2 -13500} C_VEL
LIN {X 0,Y 355.191,Z 225.238,A -85,B 0,C 180,E1 -13502.268,E2 -13502.268} C_VEL
LIN {X 0,Y 355.074,Z 225.257,A -85,B 0,C 180,E1 -13506.821,E2 -13506.821} C_VEL
LIN {X 0,Y 354.932,Z 225.271,A -85,B 0,C 180,E1 -13510.266,E2 -13510.266} C_VEL
LIN {X 0,Y 354.897,Z 225.274,A -85,B 0,C 180,E1 -13514.02,E2 -13514.02} C_VEL
LIN {X 0,Y 354.867,Z 225.279,A -85,B 0,C 180,E1 -13518.105,E2 -13518.105} C_VEL
LIN {X 0,Y 354.772,Z 225.291,A -85,B 0,C 180,E1 -13522.11,E2 -13522.11} C_VEL
LIN {X 0,Y 354.857,Z 225.279,A -85,B 0,C 180,E1 -13525.831,E2 -13525.831} C_VEL
LIN {X 0,Y 354.817,Z 225.284,A -85,B 0,C 180,E1 -13529.682,E2 -13529.682} C_VEL
LIN {X 0,Y 354.772,Z 225.29,A -85,B 0,C 180,E1 -13533.706,E2 -13533.706} C_VEL
LIN {X 0,Y 354.764,Z 225.296,A -85,B 0,C 180,E1 -13536.464,E2 -13536.464} C_VEL
LIN {X 0,Y 354.794,Z 225.287,A -85,B 0,C 180,E1 -13539.428,E2 -13539.428} C_VEL
LIN {X 0,Y 354.807,Z 225.286,A -85,B 0,C 180,E1 -13542.88,E2 -13542.88} C_VEL
LIN {X 0,Y 354.756,Z 225.297,A -85,B 0,C 180,E1 -13546.11,E2 -13546.11} C_VEL
LIN {X 0,Y 354.764,Z 225.291,A -85,B 0,C 180,E1 -13549.183,E2 -13549.183} C_VEL
LIN {X 0,Y 354.787,Z 225.291,A -85,B 0,C 180,E1 -13552.407,E2 -13552.407} C_VEL
LIN {X 0,Y 354.794,Z 225.287,A -85,B 0,C 180,E1 -13554.945,E2 -13554.945} C_VEL
LIN {X 0,Y 354.778,Z 225.291,A -85,B 0,C 180,E1 -13558.41,E2 -13558.41} C_VEL
LIN {X 0,Y 354.834,Z 225.285,A -85,B 0,C 180,E1 -13561.623,E2 -13561.623} C_VEL
LIN {X 0,Y 354.888,Z 225.279,A -85,B 0,C 180,E1 -13564.177,E2 -13564.177} C_VEL
LIN {X 0,Y 354.808,Z 225.291,A -85,B 0,C 180,E1 -13567.897,E2 -13567.897} C_VEL
LIN {X 0,Y 354.885,Z 225.281,A -85,B 0,C 180,E1 -13571.912,E2 -13571.912} C_VEL
LIN {X 0,Y 354.941,Z 225.272,A -85,B 0,C 180,E1 -13575.985,E2 -13575.985} C_VEL
LIN {X 0,Y 354.954,Z 225.377,A -85,B 0,C 180,E1 -13578.04,E2 -13578.04} C_VEL
LIN {X 0,Y 356.029,Z 230.831,A -85,B 0,C 180,E1 -13579.493,E2 -13579.493} C_VEL
LIN {X 0,Y 359.959,Z 243.475,A -85,B 0,C 180,E1 -13579.965,E2 -13579.965} C_VEL
LIN {X 0,Y 362.184,Z 256.654,A -85,B 0,C 180,E1 -13580.35,E2 -13580.35} C_VEL
LIN {X 0,Y 360.698,Z 337.473,A -85,B 0,C 180,E1 -13581.953,E2 -13581.953} C_VEL
LIN {X 0,Y 360.18,Z 350.904,A -85,B 0,C 180,E1 -13582.435,E2 -13582.435} C_VEL
LIN {X 0,Y 359.684,Z 362.491,A -85,B 0,C 180,E1 -13583.059,E2 -13583.059} C_VEL
LIN {X 0,Y 359.145,Z 373.167,A -85,B 0,C 180,E1 -13583.824,E2 -13583.824} C_VEL
LIN {X 0,Y 358.229,Z 383.953,A -85,B 0,C 180,E1 -13584.797,E2 -13584.797} C_VEL
LIN {X 0,Y 357.353,Z 393.858,A -85,B 0,C 180,E1 -13585.914,E2 -13585.914} C_VEL
LIN {X 0,Y 356.514,Z 402.963,A -85,B 0,C 180,E1 -13587.178,E2 -13587.178} C_VEL
LIN {X 0,Y 355.758,Z 411.285,A -85,B 0,C 180,E1 -13588.587,E2 -13588.587} C_VEL
LIN {X 0,Y 354.943,Z 419.44,A -85,B 0,C 180,E1 -13590.286,E2 -13590.286} C_VEL
LIN {X 0,Y 354.388,Z 425.01,A -85,B 0,C 180,E1 -13591.707,E2 -13591.707} C_VEL
LIN {X 0,Y 354.053,Z 430.434,A -85,B 0,C 180,E1 -13593.416,E2 -13593.416} C_VEL
LIN {X 0,Y 353.729,Z 434.701,A -85,B 0,C 180,E1 -13595.131,E2 -13595.131} C_VEL
LIN {X 0,Y 353.507,Z 437.911,A -85,B 0,C 180,E1 -13596.852,E2 -13596.852} C_VEL
LIN {X 0,Y 353.382,Z 439.514,A -85,B 0,C 180,E1 -13598.004,E2 -13598.004} C_VEL
LIN {X 0,Y 353.262,Z 440.707,A -85,B 0,C 180,E1 -13599.159,E2 -13599.159} C_VEL
LIN {X 0,Y 353.279,Z 441.803,A -85,B 0,C 180,E1 -13601.476,E2 -13601.476} C_VEL
LIN {X 0,Y 353.359,Z 441.689,A -85,B 0,C 180,E1 -13602.948,E2 -13602.948} C_VEL
LIN {X 0,Y 353.492,Z 440.432,A -85,B 0,C 180,E1 -13604.98,E2 -13604.98} C_VEL
LIN {X 0,Y 353.712,Z 439.136,A -85,B 0,C 180,E1 -13606.152,E2 -13606.152} C_VEL
LIN {X 0,Y 354.085,Z 436.769,A -85,B 0,C 180,E1 -13607.688,E2 -13607.688} C_VEL
LIN {X 0,Y 354.707,Z 432.494,A -85,B 0,C 180,E1 -13609.684,E2 -13609.684} C_VEL
LIN {X 0,Y 355.407,Z 427.888,A -85,B 0,C 180,E1 -13611.31,E2 -13611.31} C_VEL
LIN {X 0,Y 356.431,Z 421.008,A -85,B 0,C 180,E1 -13613.226,E2 -13613.226} C_VEL
LIN {X 0,Y 357.741,Z 412.687,A -85,B 0,C 180,E1 -13615.021,E2 -13615.021} C_VEL
LIN {X 0,Y 358.866,Z 404.48,A -85,B 0,C 180,E1 -13616.457,E2 -13616.457} C_VEL
LIN {X 0,Y 360.232,Z 394.152,A -85,B 0,C 180,E1 -13617.919,E2 -13617.919} C_VEL
LIN {X 0,Y 360.713,Z 390.444,A -85,B 0,C 180,E1 -13618.363,E2 -13618.363} C_VEL
LIN {X 0,Y 360.726,Z 385.735,A -85,B 0,C 180,E1 -13618.934,E2 -13618.934} C_VEL
LIN {X 0,Y 358.842,Z 377.979,A -85,B 0,C 180,E1 -13619.882,E2 -13619.882} C_VEL
LIN {X 0,Y 356.885,Z 369.823,A -85,B 0,C 180,E1 -13620.731,E2 -13620.731} C_VEL
LIN {X 0,Y 356.761,Z 364.492,A -85,B 0,C 180,E1 -13621.136,E2 -13621.136} C_VEL
LIN {X 0,Y 357.74,Z 351.086,A -85,B 0,C 180,E1 -13621.868,E2 -13621.868} C_VEL
LIN {X 0,Y 358.31,Z 338.524,A -85,B 0,C 180,E1 -13622.326,E2 -13622.326} C_VEL
LIN {X 0,Y 360.11,Z 258.617,A -85,B 0,C 180,E1 -13623.961,E2 -13623.961} C_VEL
LIN {X 0,Y 358.448,Z 252.89,A -85,B 0,C 180,E1 -13624.223,E2 -13624.223} C_VEL
LIN {X 0,Y 350.41,Z 234.617,A -85,B 0,C 180,E1 -13625.317,E2 -13625.317} C_VEL
LIN {X 0,Y 349.153,Z 231.779,A -85,B 0,C 180,E1 -13625.509,E2 -13625.509} C_VEL
LIN {X 0,Y 347.788,Z 226.167,A -85,B 0,C 180,E1 -13627.24,E2 -13627.24} C_VEL
LIN {X 0,Y 347.75,Z 226.164,A -85,B 0,C 180,E1 -13630.293,E2 -13630.293} C_VEL
LIN {X 0,Y 347.759,Z 226.162,A -85,B 0,C 180,E1 -13633.4,E2 -13633.4} C_VEL
LIN {X 0,Y 347.775,Z 226.166,A -85,B 0,C 180,E1 -13636.675,E2 -13636.675} C_VEL
LIN {X 0,Y 347.777,Z 226.163,A -85,B 0,C 180,E1 -13640.164,E2 -13640.164} C_VEL
LIN {X 0,Y 347.776,Z 226.167,A -85,B 0,C 180,E1 -13644.123,E2 -13644.123} C_VEL
LIN {X 0,Y 347.724,Z 226.168,A -85,B 0,C 180,E1 -13648.085,E2 -13648.085} C_VEL
LIN {X 0,Y 347.791,Z 226.162,A -85,B 0,C 180,E1 -13650.988,E2 -13650.988} C_VEL
LIN {X 0,Y 347.814,Z 226.156,A -85,B 0,C 180,E1 -13653.606,E2 -13653.606} C_VEL
LIN {X 0,Y 347.767,Z 226.158,A -85,B 0,C 180,E1 -13656.16,E2 -13656.16} C_VEL
LIN {X 0,Y 347.763,Z 226.159,A -85,B 0,C 180,E1 -13659.906,E2 -13659.906} C_VEL
LIN {X 0,Y 347.847,Z 226.154,A -85,B 0,C 180,E1 -13662.358,E2 -13662.358} C_VEL
LIN {X 0,Y 347.879,Z 226.151,A -85,B 0,C 180,E1 -13665.97,E2 -13665.97} C_VEL
LIN {X 0,Y 347.889,Z 226.145,A -85,B 0,C 180,E1 -13669.524,E2 -13669.524} C_VEL
LIN {X 0,Y 348.07,Z 226.123,A -85,B 0,C 180,E1 -13673.041,E2 -13673.041} C_VEL
LIN {X 0,Y 348.179,Z 226.106,A -85,B 0,C 180,E1 -13677.686,E2 -13677.686} C_VEL
LIN {X 0,Y 348.281,Z 226.099,A -85,B 0,C 180,E1 -13680,E2 -13680} C_VEL
LIN {X 0,Y 348.178,Z 226.108,A -85,B 0,C 180,E1 -13682.314,E2 -13682.314} C_VEL
LIN {X 0,Y 348.042,Z 226.125,A -85,B 0,C 180,E1 -13686.959,E2 -13686.959} C_VEL
LIN {X 0,Y 347.875,Z 226.151,A -85,B 0,C 180,E1 -13690.476,E2 -13690.476} C_VEL
LIN {X 0,Y 347.88,Z 226.148,A -85,B 0,C 180,E1 -13694.151,E2 -13694.151} C_VEL
LIN {X 0,Y 347.809,Z 226.156,A -85,B 0,C 180,E1 -13698.259,E2 -13698.259} C_VEL
LIN {X 0,Y 347.744,Z 226.16,A -85,B 0,C 180,E1 -13701.625,E2 -13701.625} C_VEL
LIN {X 0,Y 347.723,Z 226.163,A -85,B 0,C 180,E1 -13705.115,E2 -13705.115} C_VEL
LIN {X 0,Y 347.72,Z 226.17,A -85,B 0,C 180,E1 -13707.702,E2 -13707.702} C_VEL
LIN {X 0,Y 347.714,Z 226.166,A -85,B 0,C 180,E1 -13710.351,E2 -13710.351} C_VEL
LIN {X 0,Y 347.735,Z 226.163,A -85,B 0,C 180,E1 -13714.045,E2 -13714.045} C_VEL
LIN {X 0,Y 347.743,Z 226.156,A -85,B 0,C 180,E1 -13717.323,E2 -13717.323} C_VEL
LIN {X 0,Y 347.71,Z 226.165,A -85,B 0,C 180,E1 -13720.3,E2 -13720.3} C_VEL
LIN {X 0,Y 347.714,Z 226.17,A -85,B 0,C 180,E1 -13723.41,E2 -13723.41} C_VEL
LIN {X 0,Y 347.717,Z 226.171,A -85,B 0,C 180,E1 -13726.688,E2 -13726.688} C_VEL
LIN {X 0,Y 347.695,Z 226.177,A -85,B 0,C 180,E1 -13730.183,E2 -13730.183} C_VEL
LIN {X 0,Y 347.751,Z 226.166,A -85,B 0,C 180,E1 -13732.679,E2 -13732.679} C_VEL
LIN {X 0,Y 347.745,Z 226.173,A -85,B 0,C 180,E1 -13735.957,E2 -13735.957} C_VEL
LIN {X 0,Y 347.776,Z 226.254,A -85,B 0,C 180,E1 -13737.003,E2 -13737.003} C_VEL
LIN {X 0,Y 350.608,Z 237.835,A -85,B 0,C 180,E1 -13740.257,E2 -13740.257} C_VEL
LIN {X 0,Y 352.544,Z 247.068,A -85,B 0,C 180,E1 -13742.71,E2 -13742.71} C_VEL
LIN {X 0,Y 353.183,Z 250.395,A -85,B 0,C 180,E1 -13743.567,E2 -13743.567} C_VEL
LIN {X 0,Y 352.135,Z 260.186,A -85,B 0,C 180,E1 -13745.826,E2 -13745.826} C_VEL
LIN {X 0,Y 357.451,Z 287.424,A -85,B 0,C 180,E1 -13746.874,E2 -13746.874} C_VEL
LIN {X 0,Y 359.257,Z 299.626,A -85,B 0,C 180,E1 -13747.285,E2 -13747.285} C_VEL
LIN {X 0,Y 357.776,Z 369.421,A -85,B 0,C 180,E1 -13748.728,E2 -13748.728} C_VEL
LIN {X 0,Y 356.895,Z 383.267,A -85,B 0,C 180,E1 -13749.24,E2 -13749.24} C_VEL
LIN {X 0,Y 355.81,Z 395.688,A -85,B 0,C 180,E1 -13749.928,E2 -13749.928} C_VEL
LIN {X 0,Y 354.469,Z 406.796,A -85,B 0,C 180,E1 -13750.754,E2 -13750.754} C_VEL
LIN {X 0,Y 353.043,Z 418.349,A -85,B 0,C 180,E1 -13751.877,E2 -13751.877} C_VEL
LIN {X 0,Y 351.631,Z 428.77,A -85,B 0,C 180,E1 -13753.153,E2 -13753.153} C_VEL
LIN {X 0,Y 350.213,Z 438.276,A -85,B 0,C 180,E1 -13754.595,E2 -13754.595} C_VEL
LIN {X 0,Y 349.009,Z 447.288,A -85,B 0,C 180,E1 -13756.313,E2 -13756.313} C_VEL
LIN {X 0,Y 347.852,Z 454.647,A -85,B 0,C 180,E1 -13758.047,E2 -13758.047} C_VEL
LIN {X 0,Y 346.998,Z 461.442,A -85,B 0,C 180,E1 -13760.086,E2 -13760.086} C_VEL
LIN {X 0,Y 346.523,Z 465.952,A -85,B 0,C 180,E1 -13761.837,E2 -13761.837} C_VEL
LIN {X 0,Y 346.243,Z 470.103,A -85,B 0,C 180,E1 -13764.042,E2 -13764.042} C_VEL
LIN {X 0,Y 346.194,Z 471.861,A -85,B 0,C 180,E1 -13765.341,E2 -13765.341} C_VEL
LIN {X 0,Y 346.163,Z 472.965,A -85,B 0,C 180,E1 -13766.506,E2 -13766.506} C_VEL
LIN {X 0,Y 346.258,Z 473.998,A -85,B 0,C 180,E1 -13768.835,E2 -13768.835} C_VEL
LIN {X 0,Y 346.319,Z 473.933,A -85,B 0,C 180,E1 -13769.998,E2 -13769.998} C_VEL
LIN {X 0,Y 346.297,Z 473.432,A -85,B 0,C 180,E1 -13771.161,E2 -13771.161} C_VEL
LIN {X 0,Y 346.194,Z 471.207,A -85,B 0,C 180,E1 -13773.489,E2 -13773.489} C_VEL
LIN {X 0,Y 346.223,Z 468.414,A -85,B 0,C 180,E1 -13775.238,E2 -13775.238} C_VEL
LIN {X 0,Y 346.339,Z 464.578,A -85,B 0,C 180,E1 -13776.99,E2 -13776.99} C_VEL
LIN {X 0,Y 346.566,Z 459.595,A -85,B 0,C 180,E1 -13778.745,E2 -13778.745} C_VEL
LIN {X 0,Y 346.975,Z 453.313,A -85,B 0,C 180,E1 -13780.5,E2 -13780.5} C_VEL
LIN {X 0,Y 347.718,Z 445.468,A -85,B 0,C 180,E1 -13782.249,E2 -13782.249} C_VEL
LIN {X 0,Y 348.48,Z 437.429,A -85,B 0,C 180,E1 -13783.704,E2 -13783.704} C_VEL
LIN {X 0,Y 349.413,Z 427.61,A -85,B 0,C 180,E1 -13785.154,E2 -13785.154} C_VEL
LIN {X 0,Y 350.345,Z 416.675,A -85,B 0,C 180,E1 -13786.456,E2 -13786.456} C_VEL
LIN {X 0,Y 351.386,Z 406.013,A -85,B 0,C 180,E1 -13787.454,E2 -13787.454} C_VEL
LIN {X 0,Y 352.268,Z 394.276,A -85,B 0,C 180,E1 -13788.31,E2 -13788.31} C_VEL
LIN {X 0,Y 353.155,Z 380.99,A -85,B 0,C 180,E1 -13789.014,E2 -13789.014} C_VEL
LIN {X 0,Y 353.7,Z 368.937,A -85,B 0,C 180,E1 -13789.436,E2 -13789.436} C_VEL
LIN {X 0,Y 354.77,Z 297.852,A -85,B 0,C 180,E1 -13790.886,E2 -13790.886} C_VEL
LIN {X 0,Y 349.815,Z 260.873,A -85,B 0,C 180,E1 -13791.928,E2 -13791.928} C_VEL
LIN {X 0,Y 351.212,Z 245.395,A -85,B 0,C 180,E1 -13795.373,E2 -13795.373} C_VEL
LIN {X 0,Y 351.04,Z 242.145,A -85,B 0,C 180,E1 -13796.128,E2 -13796.128} C_VEL
LIN {X 0,Y 348.815,Z 230.767,A -85,B 0,C 180,E1 -13798.912,E2 -13798.912} C_VEL
LIN {X 0,Y 347.82,Z 226.162,A -85,B 0,C 180,E1 -13800.101,E2 -13800.101} C_VEL
LIN {X 0,Y 347.726,Z 226.169,A -85,B 0,C 180,E1 -13804.459,E2 -13804.459} C_VEL
LIN {X 0,Y 347.752,Z 226.17,A -85,B 0,C 180,E1 -13807.984,E2 -13807.984} C_VEL
LIN {X 0,Y 347.726,Z 226.173,A -85,B 0,C 180,E1 -13811.826,E2 -13811.826} C_VEL
LIN {X 0,Y 347.749,Z 226.165,A -85,B 0,C 180,E1 -13815.011,E2 -13815.011} C_VEL
LIN {X 0,Y 347.757,Z 226.164,A -85,B 0,C 180,E1 -13818.386,E2 -13818.386} C_VEL
LIN {X 0,Y 347.743,Z 226.168,A -85,B 0,C 180,E1 -13822.007,E2 -13822.007} C_VEL
LIN {X 0,Y 347.709,Z 226.174,A -85,B 0,C 180,E1 -13825.532,E2 -13825.532} C_VEL
LIN {X 0,Y 347.726,Z 226.173,A -85,B 0,C 180,E1 -13829.65,E2 -13829.65} C_VEL
LIN {X 0,Y 347.812,Z 226.157,A -85,B 0,C 180,E1 -13832.742,E2 -13832.742} C_VEL
LIN {X 0,Y 347.775,Z 226.162,A -85,B 0,C 180,E1 -13836.161,E2 -13836.161} C_VEL
LIN {X 0,Y 347.8,Z 226.16,A -85,B 0,C 180,E1 -13839.909,E2 -13839.909} C_VEL
LIN {X 0,Y 347.822,Z 226.155,A -85,B 0,C 180,E1 -13842.357,E2 -13842.357} C_VEL
LIN {X 0,Y 347.853,Z 226.152,A -85,B 0,C 180,E1 -13845.969,E2 -13845.969} C_VEL
LIN {X 0,Y 347.885,Z 226.151,A -85,B 0,C 180,E1 -13849.524,E2 -13849.524} C_VEL
LIN {X 0,Y 348.066,Z 226.13,A -85,B 0,C 180,E1 -13853.042,E2 -13853.042} C_VEL
LIN {X 0,Y 348.159,Z 226.114,A -85,B 0,C 180,E1 -13857.686,E2 -13857.686} C_VEL
LIN {X 0,Y 348.276,Z 226.099,A -85,B 0,C 180,E1 -13860,E2 -13860} C_VEL
LIN {X 0,Y 348.154,Z 226.115,A -85,B 0,C 180,E1 -13862.314,E2 -13862.314} C_VEL
LIN {X 0,Y 348.041,Z 226.134,A -85,B 0,C 180,E1 -13866.959,E2 -13866.959} C_VEL
LIN {X 0,Y 347.883,Z 226.15,A -85,B 0,C 180,E1 -13870.476,E2 -13870.476} C_VEL
LIN {X 0,Y 347.855,Z 226.152,A -85,B 0,C 180,E1 -13874.152,E2 -13874.152} C_VEL
LIN {X 0,Y 347.801,Z 226.16,A -85,B 0,C 180,E1 -13878.269,E2 -13878.269} C_VEL
LIN {X 0,Y 347.724,Z 226.168,A -85,B 0,C 180,E1 -13881.628,E2 -13881.628} C_VEL
LIN {X 0,Y 347.77,Z 226.163,A -85,B 0,C 180,E1 -13885.112,E2 -13885.112} C_VEL
LIN {X 0,Y 347.772,Z 226.162,A -85,B 0,C 180,E1 -13887.697,E2 -13887.697} C_VEL
LIN {X 0,Y 347.727,Z 226.172,A -85,B 0,C 180,E1 -13890.35,E2 -13890.35} C_VEL
LIN {X 0,Y 347.71,Z 226.175,A -85,B 0,C 180,E1 -13894.468,E2 -13894.468} C_VEL
LIN {X 0,Y 347.742,Z 226.168,A -85,B 0,C 180,E1 -13897.993,E2 -13897.993} C_VEL
LIN {X 0,Y 347.757,Z 226.164,A -85,B 0,C 180,E1 -13901.614,E2 -13901.614} C_VEL
LIN {X 0,Y 347.749,Z 226.165,A -85,B 0,C 180,E1 -13905.02,E2 -13905.02} C_VEL
LIN {X 0,Y 347.727,Z 226.171,A -85,B 0,C 180,E1 -13908.402,E2 -13908.402} C_VEL
LIN {X 0,Y 347.753,Z 226.169,A -85,B 0,C 180,E1 -13912.016,E2 -13912.016} C_VEL
LIN {X 0,Y 347.727,Z 226.169,A -85,B 0,C 180,E1 -13915.541,E2 -13915.541} C_VEL
LIN {X 0,Y 347.73,Z 226.17,A -85,B 0,C 180,E1 -13918.305,E2 -13918.305} C_VEL
LIN {X 0,Y 347.766,Z 226.162,A -85,B 0,C 180,E1 -13920.992,E2 -13920.992} C_VEL
LIN {X 0,Y 347.82,Z 226.159,A -85,B 0,C 180,E1 -13923.612,E2 -13923.612} C_VEL
LIN {X 0,Y 347.776,Z 226.164,A -85,B 0,C 180,E1 -13926.166,E2 -13926.166} C_VEL
LIN {X 0,Y 347.793,Z 226.164,A -85,B 0,C 180,E1 -13929.913,E2 -13929.913} C_VEL
LIN {X 0,Y 347.828,Z 226.159,A -85,B 0,C 180,E1 -13933.572,E2 -13933.572} C_VEL
LIN {X 0,Y 347.888,Z 226.149,A -85,B 0,C 180,E1 -13937.164,E2 -13937.164} C_VEL
LIN {X 0,Y 347.887,Z 226.175,A -85,B 0,C 180,E1 -13937.757,E2 -13937.757} C_VEL
LIN {X 0,Y 348.896,Z 231.121,A -85,B 0,C 180,E1 -13939.103,E2 -13939.103} C_VEL
LIN {X 0,Y 353.317,Z 244.96,A -85,B 0,C 180,E1 -13939.647,E2 -13939.647} C_VEL
LIN {X 0,Y 355.406,Z 257.628,A -85,B 0,C 180,E1 -13940.024,E2 -13940.024} C_VEL
LIN {X 0,Y 353.895,Z 338.103,A -85,B 0,C 180,E1 -13941.653,E2 -13941.653} C_VEL
LIN {X 0,Y 353.357,Z 351.409,A -85,B 0,C 180,E1 -13942.144,E2 -13942.144} C_VEL
LIN {X 0,Y 352.816,Z 362.958,A -85,B 0,C 180,E1 -13942.779,E2 -13942.779} C_VEL
LIN {X 0,Y 352.267,Z 373.599,A -85,B 0,C 180,E1 -13943.559,E2 -13943.559} C_VEL
LIN {X 0,Y 351.317,Z 384.366,A -85,B 0,C 180,E1 -13944.55,E2 -13944.55} C_VEL
LIN {X 0,Y 350.412,Z 394.257,A -85,B 0,C 180,E1 -13945.689,E2 -13945.689} C_VEL
LIN {X 0,Y 349.432,Z 404.238,A -85,B 0,C 180,E1 -13947.12,E2 -13947.12} C_VEL
LIN {X 0,Y 348.524,Z 413.883,A -85,B 0,C 180,E1 -13948.847,E2 -13948.847} C_VEL
LIN {X 0,Y 347.685,Z 421.612,A -85,B 0,C 180,E1 -13950.581,E2 -13950.581} C_VEL
LIN {X 0,Y 347.211,Z 427.785,A -85,B 0,C 180,E1 -13952.322,E2 -13952.322} C_VEL
LIN {X 0,Y 346.77,Z 432.711,A -85,B 0,C 180,E1 -13954.069,E2 -13954.069} C_VEL
LIN {X 0,Y 346.552,Z 436.513,A -85,B 0,C 180,E1 -13955.821,E2 -13955.821} C_VEL
LIN {X 0,Y 346.398,Z 438.483,A -85,B 0,C 180,E1 -13956.994,E2 -13956.994} C_VEL
LIN {X 0,Y 346.281,Z 440.04,A -85,B 0,C 180,E1 -13958.169,E2 -13958.169} C_VEL
LIN {X 0,Y 346.16,Z 441.148,A -85,B 0,C 180,E1 -13959.349,E2 -13959.349} C_VEL
LIN {X 0,Y 346.193,Z 442.156,A -85,B 0,C 180,E1 -13961.714,E2 -13961.714} C_VEL
LIN {X 0,Y 346.269,Z 442.027,A -85,B 0,C 180,E1 -13963.035,E2 -13963.035} C_VEL
LIN {X 0,Y 346.477,Z 440.609,A -85,B 0,C 180,E1 -13965.29,E2 -13965.29} C_VEL
LIN {X 0,Y 346.7,Z 439.269,A -85,B 0,C 180,E1 -13966.488,E2 -13966.488} C_VEL
LIN {X 0,Y 347.053,Z 437.151,A -85,B 0,C 180,E1 -13967.865,E2 -13967.865} C_VEL
LIN {X 0,Y 347.809,Z 432.437,A -85,B 0,C 180,E1 -13970.091,E2 -13970.091} C_VEL
LIN {X 0,Y 348.723,Z 426.861,A -85,B 0,C 180,E1 -13972.018,E2 -13972.018} C_VEL
LIN {X 0,Y 349.904,Z 419.409,A -85,B 0,C 180,E1 -13974,E2 -13974} C_VEL
LIN {X 0,Y 351.156,Z 411.723,A -85,B 0,C 180,E1 -13975.623,E2 -13975.623} C_VEL
LIN {X 0,Y 352.292,Z 403.831,A -85,B 0,C 180,E1 -13976.99,E2 -13976.99} C_VEL
LIN {X 0,Y 353.593,Z 394.401,A -85,B 0,C 180,E1 -13978.329,E2 -13978.329} C_VEL
LIN {X 0,Y 354.962,Z 384.012,A -85,B 0,C 180,E1 -13979.507,E2 -13979.507} C_VEL
LIN {X 0,Y 356.131,Z 372.614,A -85,B 0,C 180,E1 -13980.54,E2 -13980.54} C_VEL
LIN {X 0,Y 356.761,Z 364.492,A -85,B 0,C 180,E1 -13981.136,E2 -13981.136} C_VEL
LIN {X 0,Y 356.692,Z 359.049,A -85,B 0,C 180,E1 -13981.504,E2 -13981.504} C_VEL
LIN {X 0,Y 353.741,Z 346.625,A -85,B 0,C 180,E1 -13982.38,E2 -13982.38} C_VEL
LIN {X 0,Y 352.259,Z 339.248,A -85,B 0,C 180,E1 -13982.77,E2 -13982.77} C_VEL
LIN {X 0,Y 352.019,Z 335.4,A -85,B 0,C 180,E1 -13982.895,E2 -13982.895} C_VEL
LIN {X 0,Y 353.785,Z 259.723,A -85,B 0,C 180,E1 -13984.456,E2 -13984.456} C_VEL
LIN {X 0,Y 351.415,Z 253.028,A -85,B 0,C 180,E1 -13984.808,E2 -13984.808} C_VEL
LIN {X 0,Y 343.53,Z 235.48,A -85,B 0,C 180,E1 -13985.917,E2 -13985.917} C_VEL
LIN {X 0,Y 341.953,Z 232.114,A -85,B 0,C 180,E1 -13986.168,E2 -13986.168} C_VEL
LIN {X 0,Y 340.749,Z 227.044,A -85,B 0,C 180,E1 -13987.755,E2 -13987.755} C_VEL
LIN {X 0,Y 340.699,Z 227.048,A -85,B 0,C 180,E1 -13991.306,E2 -13991.306} C_VEL
LIN {X 0,Y 340.708,Z 227.037,A -85,B 0,C 180,E1 -13994.532,E2 -13994.532} C_VEL
LIN {X 0,Y 340.739,Z 227.042,A -85,B 0,C 180,E1 -13997.944,E2 -13997.944} C_VEL
LIN {X 0,Y 340.725,Z 227.042,A -85,B 0,C 180,E1 -14000.251,E2 -14000.251} C_VEL
LIN {X 0,Y 340.699,Z 227.044,A -85,B 0,C 180,E1 -14003.558,E2 -14003.558} C_VEL
LIN {X 0,Y 340.68,Z 227.046,A -85,B 0,C 180,E1 -14006.152,E2 -14006.152} C_VEL
LIN {X 0,Y 340.761,Z 227.039,A -85,B 0,C 180,E1 -14010.331,E2 -14010.331} C_VEL
LIN {X 0,Y 340.789,Z 227.027,A -85,B 0,C 180,E1 -14013.018,E2 -14013.018} C_VEL
LIN {X 0,Y 340.738,Z 227.037,A -85,B 0,C 180,E1 -14015.637,E2 -14015.637} C_VEL
LIN {X 0,Y 340.699,Z 227.043,A -85,B 0,C 180,E1 -14019.471,E2 -14019.471} C_VEL
LIN {X 0,Y 340.829,Z 227.03,A -85,B 0,C 180,E1 -14021.982,E2 -14021.982} C_VEL
LIN {X 0,Y 340.834,Z 227.026,A -85,B 0,C 180,E1 -14025.716,E2 -14025.716} C_VEL
LIN {X 0,Y 340.836,Z 227.022,A -85,B 0,C 180,E1 -14029.305,E2 -14029.305} C_VEL
LIN {X 0,Y 341.039,Z 227,A -85,B 0,C 180,E1 -14032.897,E2 -14032.897} C_VEL
LIN {X 0,Y 341.141,Z 226.982,A -85,B 0,C 180,E1 -14037.638,E2 -14037.638} C_VEL
LIN {X 0,Y 341.232,Z 226.977,A -85,B 0,C 180,E1 -14040,E2 -14040} C_VEL
LIN {X 0,Y 341.14,Z 226.985,A -85,B 0,C 180,E1 -14042.361,E2 -14042.361} C_VEL
LIN {X 0,Y 340.988,Z 227.002,A -85,B 0,C 180,E1 -14047.104,E2 -14047.104} C_VEL
LIN {X 0,Y 340.827,Z 227.031,A -85,B 0,C 180,E1 -14050.695,E2 -14050.695} C_VEL
LIN {X 0,Y 340.845,Z 227.025,A -85,B 0,C 180,E1 -14054.326,E2 -14054.326} C_VEL
LIN {X 0,Y 340.765,Z 227.034,A -85,B 0,C 180,E1 -14058.44,E2 -14058.44} C_VEL
LIN {X 0,Y 340.701,Z 227.037,A -85,B 0,C 180,E1 -14061.843,E2 -14061.843} C_VEL
LIN {X 0,Y 340.659,Z 227.041,A -85,B 0,C 180,E1 -14065.674,E2 -14065.674} C_VEL
LIN {X 0,Y 340.666,Z 227.052,A -85,B 0,C 180,E1 -14068.326,E2 -14068.326} C_VEL
LIN {X 0,Y 340.667,Z 227.05,A -85,B 0,C 180,E1 -14071.048,E2 -14071.048} C_VEL
LIN {X 0,Y 340.702,Z 227.044,A -85,B 0,C 180,E1 -14075.281,E2 -14075.281} C_VEL
LIN {X 0,Y 340.682,Z 227.026,A -85,B 0,C 180,E1 -14078.384,E2 -14078.384} C_VEL
LIN {X 0,Y 340.689,Z 227.048,A -85,B 0,C 180,E1 -14082.046,E2 -14082.046} C_VEL
LIN {X 0,Y 340.643,Z 227.055,A -85,B 0,C 180,E1 -14086.229,E2 -14086.229} C_VEL
LIN {X 0,Y 340.664,Z 227.041,A -85,B 0,C 180,E1 -14088.689,E2 -14088.689} C_VEL
LIN {X 0,Y 340.713,Z 227.037,A -85,B 0,C 180,E1 -14091.772,E2 -14091.772} C_VEL
LIN {X 0,Y 340.72,Z 227.044,A -85,B 0,C 180,E1 -14095.596,E2 -14095.596} C_VEL
LIN {X 0,Y 340.736,Z 227.195,A -85,B 0,C 180,E1 -14096.47,E2 -14096.47} C_VEL
LIN {X 0,Y 343.395,Z 237.99,A -85,B 0,C 180,E1 -14099.597,E2 -14099.597} C_VEL
LIN {X 0,Y 345.411,Z 247.093,A -85,B 0,C 180,E1 -14102.098,E2 -14102.098} C_VEL
LIN {X 0,Y 346.32,Z 252.366,A -85,B 0,C 180,E1 -14103.484,E2 -14103.484} C_VEL
LIN {X 0,Y 345.462,Z 259.831,A -85,B 0,C 180,E1 -14105.239,E2 -14105.239} C_VEL
LIN {X 0,Y 350.866,Z 287.218,A -85,B 0,C 180,E1 -14106.334,E2 -14106.334} C_VEL
LIN {X 0,Y 352.88,Z 301.133,A -85,B 0,C 180,E1 -14106.813,E2 -14106.813} C_VEL
LIN {X 0,Y 351.34,Z 369.097,A -85,B 0,C 180,E1 -14108.242,E2 -14108.242} C_VEL
LIN {X 0,Y 350.443,Z 382.931,A -85,B 0,C 180,E1 -14108.762,E2 -14108.762} C_VEL
LIN {X 0,Y 349.318,Z 395.346,A -85,B 0,C 180,E1 -14109.462,E2 -14109.462} C_VEL
LIN {X 0,Y 347.805,Z 407.241,A -85,B 0,C 180,E1 -14110.37,E2 -14110.37} C_VEL
LIN {X 0,Y 346.302,Z 418.649,A -85,B 0,C 180,E1 -14111.512,E2 -14111.512} C_VEL
LIN {X 0,Y 344.831,Z 428.962,A -85,B 0,C 180,E1 -14112.81,E2 -14112.81} C_VEL
LIN {X 0,Y 343.284,Z 438.888,A -85,B 0,C 180,E1 -14114.377,E2 -14114.377} C_VEL
LIN {X 0,Y 342.104,Z 447.288,A -85,B 0,C 180,E1 -14116.031,E2 -14116.031} C_VEL
LIN {X 0,Y 340.863,Z 454.589,A -85,B 0,C 180,E1 -14117.798,E2 -14117.798} C_VEL
LIN {X 0,Y 339.973,Z 461.309,A -85,B 0,C 180,E1 -14119.879,E2 -14119.879} C_VEL
LIN {X 0,Y 339.463,Z 465.773,A -85,B 0,C 180,E1 -14121.666,E2 -14121.666} C_VEL
LIN {X 0,Y 339.269,Z 468.142,A -85,B 0,C 180,E1 -14122.859,E2 -14122.859} C_VEL
LIN {X 0,Y 339.137,Z 470.173,A -85,B 0,C 180,E1 -14124.108,E2 -14124.108} C_VEL
LIN {X 0,Y 339.095,Z 471.607,A -85,B 0,C 180,E1 -14125.243,E2 -14125.243} C_VEL
LIN {X 0,Y 339.087,Z 472.685,A -85,B 0,C 180,E1 -14126.433,E2 -14126.433} C_VEL
LIN {X 0,Y 339.16,Z 473.679,A -85,B 0,C 180,E1 -14128.811,E2 -14128.811} C_VEL
LIN {X 0,Y 339.226,Z 473.589,A -85,B 0,C 180,E1 -14129.998,E2 -14129.998} C_VEL
LIN {X 0,Y 339.2,Z 473.057,A -85,B 0,C 180,E1 -14131.185,E2 -14131.185} C_VEL
LIN {X 0,Y 339.118,Z 470.794,A -85,B 0,C 180,E1 -14133.562,E2 -14133.562} C_VEL
LIN {X 0,Y 339.133,Z 467.694,A -85,B 0,C 180,E1 -14135.495,E2 -14135.495} C_VEL
LIN {X 0,Y 339.265,Z 464.079,A -85,B 0,C 180,E1 -14137.137,E2 -14137.137} C_VEL
LIN {X 0,Y 339.512,Z 459.046,A -85,B 0,C 180,E1 -14138.928,E2 -14138.928} C_VEL
LIN {X 0,Y 339.926,Z 452.708,A -85,B 0,C 180,E1 -14140.721,E2 -14140.721} C_VEL
LIN {X 0,Y 340.742,Z 444.772,A -85,B 0,C 180,E1 -14142.504,E2 -14142.504} C_VEL
LIN {X 0,Y 341.559,Z 436.662,A -85,B 0,C 180,E1 -14143.987,E2 -14143.987} C_VEL
LIN {X 0,Y 342.409,Z 427.792,A -85,B 0,C 180,E1 -14145.325,E2 -14145.325} C_VEL
LIN {X 0,Y 343.358,Z 417.015,A -85,B 0,C 180,E1 -14146.648,E2 -14146.648} C_VEL
LIN {X 0,Y 344.407,Z 406.559,A -85,B 0,C 180,E1 -14147.666,E2 -14147.666} C_VEL
LIN {X 0,Y 345.313,Z 395.103,A -85,B 0,C 180,E1 -14148.538,E2 -14148.538} C_VEL
LIN {X 0,Y 346.282,Z 381.455,A -85,B 0,C 180,E1 -14149.291,E2 -14149.291} C_VEL
LIN {X 0,Y 346.875,Z 368.647,A -85,B 0,C 180,E1 -14149.757,E2 -14149.757} C_VEL
LIN {X 0,Y 347.912,Z 297.803,A -85,B 0,C 180,E1 -14151.234,E2 -14151.234} C_VEL
LIN {X 0,Y 342.919,Z 260.559,A -85,B 0,C 180,E1 -14152.307,E2 -14152.307} C_VEL
LIN {X 0,Y 344.186,Z 246.997,A -85,B 0,C 180,E1 -14155.387,E2 -14155.387} C_VEL
LIN {X 0,Y 344.034,Z 243.144,A -85,B 0,C 180,E1 -14156.298,E2 -14156.298} C_VEL
LIN {X 0,Y 341.382,Z 229.99,A -85,B 0,C 180,E1 -14159.604,E2 -14159.604} C_VEL
LIN {X 0,Y 340.747,Z 227.042,A -85,B 0,C 180,E1 -14160.391,E2 -14160.391} C_VEL
LIN {X 0,Y 340.705,Z 227.045,A -85,B 0,C 180,E1 -14164.4,E2 -14164.4} C_VEL
LIN {X 0,Y 340.688,Z 227.046,A -85,B 0,C 180,E1 -14168.381,E2 -14168.381} C_VEL
LIN {X 0,Y 340.675,Z 227.05,A -85,B 0,C 180,E1 -14172.041,E2 -14172.041} C_VEL
LIN {X 0,Y 340.685,Z 227.047,A -85,B 0,C 180,E1 -14176.212,E2 -14176.212} C_VEL
LIN {X 0,Y 340.734,Z 227.044,A -85,B 0,C 180,E1 -14179.734,E2 -14179.734} C_VEL
LIN {X 0,Y 340.677,Z 227.05,A -85,B 0,C 180,E1 -14183.556,E2 -14183.556} C_VEL
LIN {X 0,Y 340.657,Z 227.049,A -85,B 0,C 180,E1 -14186.149,E2 -14186.149} C_VEL
LIN {X 0,Y 340.737,Z 227.038,A -85,B 0,C 180,E1 -14190.329,E2 -14190.329} C_VEL
LIN {X 0,Y 340.765,Z 227.036,A -85,B 0,C 180,E1 -14193.017,E2 -14193.017} C_VEL
LIN {X 0,Y 340.749,Z 227.038,A -85,B 0,C 180,E1 -14196.929,E2 -14196.929} C_VEL
LIN {X 0,Y 340.763,Z 227.036,A -85,B 0,C 180,E1 -14200.732,E2 -14200.732} C_VEL
LIN {X 0,Y 340.742,Z 227.042,A -85,B 0,C 180,E1 -14203.216,E2 -14203.216} C_VEL
LIN {X 0,Y 340.8,Z 227.032,A -85,B 0,C 180,E1 -14206.889,E2 -14206.889} C_VEL
LIN {X 0,Y 340.884,Z 227.02,A -85,B 0,C 180,E1 -14210.507,E2 -14210.507} C_VEL
LIN {X 0,Y 341.035,Z 227.004,A -85,B 0,C 180,E1 -14212.897,E2 -14212.897} C_VEL
LIN {X 0,Y 341.121,Z 226.991,A -85,B 0,C 180,E1 -14217.639,E2 -14217.639} C_VEL
LIN {X 0,Y 341.227,Z 226.976,A -85,B 0,C 180,E1 -14220,E2 -14220} C_VEL
LIN {X 0,Y 341.116,Z 226.99,A -85,B 0,C 180,E1 -14222.362,E2 -14222.362} C_VEL
LIN {X 0,Y 341.01,Z 227.008,A -85,B 0,C 180,E1 -14227.103,E2 -14227.103} C_VEL
LIN {X 0,Y 340.826,Z 227.031,A -85,B 0,C 180,E1 -14230.695,E2 -14230.695} C_VEL
LIN {X 0,Y 340.82,Z 227.028,A -85,B 0,C 180,E1 -14234.327,E2 -14234.327} C_VEL
LIN {X 0,Y 340.754,Z 227.039,A -85,B 0,C 180,E1 -14238.448,E2 -14238.448} C_VEL
LIN {X 0,Y 340.677,Z 227.046,A -85,B 0,C 180,E1 -14241.845,E2 -14241.845} C_VEL
LIN {X 0,Y 340.732,Z 227.039,A -85,B 0,C 180,E1 -14245.668,E2 -14245.668} C_VEL
LIN {X 0,Y 340.703,Z 227.046,A -85,B 0,C 180,E1 -14248.323,E2 -14248.323} C_VEL
LIN {X 0,Y 340.667,Z 227.048,A -85,B 0,C 180,E1 -14251.048,E2 -14251.048} C_VEL
LIN {X 0,Y 340.684,Z 227.045,A -85,B 0,C 180,E1 -14255.283,E2 -14255.283} C_VEL
LIN {X 0,Y 340.681,Z 227.051,A -85,B 0,C 180,E1 -14258.39,E2 -14258.39} C_VEL
LIN {X 0,Y 340.698,Z 227.043,A -85,B 0,C 180,E1 -14261.308,E2 -14261.308} C_VEL
LIN {X 0,Y 340.681,Z 227.047,A -85,B 0,C 180,E1 -14264.54,E2 -14264.54} C_VEL
LIN {X 0,Y 340.663,Z 227.049,A -85,B 0,C 180,E1 -14268.695,E2 -14268.695} C_VEL
LIN {X 0,Y 340.713,Z 227.043,A -85,B 0,C 180,E1 -14271.777,E2 -14271.777} C_VEL
LIN {X 0,Y 340.706,Z 227.044,A -85,B 0,C 180,E1 -14275.6,E2 -14275.6} C_VEL
LIN {X 0,Y 340.683,Z 227.045,A -85,B 0,C 180,E1 -14278.96,E2 -14278.96} C_VEL
LIN {X 0,Y 340.792,Z 227.031,A -85,B 0,C 180,E1 -14283.024,E2 -14283.024} C_VEL
LIN {X 0,Y 340.745,Z 227.04,A -85,B 0,C 180,E1 -14285.643,E2 -14285.643} C_VEL
LIN {X 0,Y 340.723,Z 227.042,A -85,B 0,C 180,E1 -14289.477,E2 -14289.477} C_VEL
LIN {X 0,Y 340.787,Z 227.036,A -85,B 0,C 180,E1 -14291.985,E2 -14291.985} C_VEL
LIN {X 0,Y 340.867,Z 227.028,A -85,B 0,C 180,E1 -14295.709,E2 -14295.709} C_VEL
LIN {X 0,Y 340.86,Z 227.115,A -85,B 0,C 180,E1 -14297.5,E2 -14297.5} C_VEL
LIN {X 0,Y 341.724,Z 231.436,A -85,B 0,C 180,E1 -14298.698,E2 -14298.698} C_VEL
LIN {X 0,Y 346.769,Z 247.03,A -85,B 0,C 180,E1 -14299.335,E2 -14299.335} C_VEL
LIN {X 0,Y 348.647,Z 258.002,A -85,B 0,C 180,E1 -14299.673,E2 -14299.673} C_VEL
LIN {X 0,Y 347.081,Z 338.727,A -85,B 0,C 180,E1 -14301.341,E2 -14301.341} C_VEL
LIN {X 0,Y 346.529,Z 351.922,A -85,B 0,C 180,E1 -14301.841,E2 -14301.841} C_VEL
LIN {X 0,Y 345.958,Z 363.426,A -85,B 0,C 180,E1 -14302.489,E2 -14302.489} C_VEL
LIN {X 0,Y 345.388,Z 374.034,A -85,B 0,C 180,E1 -14303.284,E2 -14303.284} C_VEL
LIN {X 0,Y 344.412,Z 384.779,A -85,B 0,C 180,E1 -14304.294,E2 -14304.294} C_VEL
LIN {X 0,Y 343.475,Z 394.651,A -85,B 0,C 180,E1 -14305.455,E2 -14305.455} C_VEL
LIN {X 0,Y 342.567,Z 403.73,A -85,B 0,C 180,E1 -14306.768,E2 -14306.768} C_VEL
LIN {X 0,Y 341.76,Z 412.035,A -85,B 0,C 180,E1 -14308.235,E2 -14308.235} C_VEL
LIN {X 0,Y 340.871,Z 420.178,A -85,B 0,C 180,E1 -14310.002,E2 -14310.002} C_VEL
LIN {X 0,Y 340.212,Z 426.735,A -85,B 0,C 180,E1 -14311.778,E2 -14311.778} C_VEL
LIN {X 0,Y 339.819,Z 431.954,A -85,B 0,C 180,E1 -14313.559,E2 -14313.559} C_VEL
LIN {X 0,Y 339.541,Z 436.021,A -85,B 0,C 180,E1 -14315.346,E2 -14315.346} C_VEL
LIN {X 0,Y 339.305,Z 439.048,A -85,B 0,C 180,E1 -14317.141,E2 -14317.141} C_VEL
LIN {X 0,Y 339.174,Z 440.536,A -85,B 0,C 180,E1 -14318.341,E2 -14318.341} C_VEL
LIN {X 0,Y 339.042,Z 442.241,A -85,B 0,C 180,E1 -14320.753,E2 -14320.753} C_VEL
LIN {X 0,Y 339.107,Z 442.509,A -85,B 0,C 180,E1 -14321.962,E2 -14321.962} C_VEL
LIN {X 0,Y 339.204,Z 442.345,A -85,B 0,C 180,E1 -14323.175,E2 -14323.175} C_VEL
LIN {X 0,Y 339.287,Z 441.767,A -85,B 0,C 180,E1 -14324.394,E2 -14324.394} C_VEL
LIN {X 0,Y 339.438,Z 440.789,A -85,B 0,C 180,E1 -14325.615,E2 -14325.615} C_VEL
LIN {X 0,Y 339.711,Z 439.396,A -85,B 0,C 180,E1 -14326.837,E2 -14326.837} C_VEL
LIN {X 0,Y 340.23,Z 436.432,A -85,B 0,C 180,E1 -14328.674,E2 -14328.674} C_VEL
LIN {X 0,Y 340.897,Z 432.367,A -85,B 0,C 180,E1 -14330.517,E2 -14330.517} C_VEL
LIN {X 0,Y 341.899,Z 426.57,A -85,B 0,C 180,E1 -14332.503,E2 -14332.503} C_VEL
LIN {X 0,Y 343.192,Z 419.065,A -85,B 0,C 180,E1 -14334.499,E2 -14334.499} C_VEL
LIN {X 0,Y 344.529,Z 411.17,A -85,B 0,C 180,E1 -14336.161,E2 -14336.161} C_VEL
LIN {X 0,Y 346.024,Z 401.135,A -85,B 0,C 180,E1 -14337.849,E2 -14337.849} C_VEL
LIN {X 0,Y 347.526,Z 390.818,A -85,B 0,C 180,E1 -14339.23,E2 -14339.23} C_VEL
LIN {X 0,Y 348.94,Z 379.738,A -85,B 0,C 180,E1 -14340.4,E2 -14340.4} C_VEL
LIN {X 0,Y 350.084,Z 366.885,A -85,B 0,C 180,E1 -14341.463,E2 -14341.463} C_VEL
LIN {X 0,Y 351.113,Z 354.434,A -85,B 0,C 180,E1 -14342.203,E2 -14342.203} C_VEL
LIN {X 0,Y 351.815,Z 341.005,A -85,B 0,C 180,E1 -14342.743,E2 -14342.743} C_VEL
LIN {X 0,Y 352.019,Z 335.4,A -85,B 0,C 180,E1 -14342.895,E2 -14342.895} C_VEL
LIN {X 0,Y 351.522,Z 329.617,A -85,B 0,C 180,E1 -14343.08,E2 -14343.08} C_VEL
LIN {X 0,Y 346.771,Z 310.986,A -85,B 0,C 180,E1 -14343.883,E2 -14343.883} C_VEL
LIN {X 0,Y 346.317,Z 305.185,A -85,B 0,C 180,E1 -14344.051,E2 -14344.051} C_VEL
LIN {X 0,Y 347.502,Z 261.367,A -85,B 0,C 180,E1 -14344.956,E2 -14344.956} C_VEL
LIN {X 0,Y 344.545,Z 253.63,A -85,B 0,C 180,E1 -14345.398,E2 -14345.398} C_VEL
LIN {X 0,Y 337.811,Z 238.821,A -85,B 0,C 180,E1 -14346.375,E2 -14346.375} C_VEL
LIN {X 0,Y 334.832,Z 232.511,A -85,B 0,C 180,E1 -14346.837,E2 -14346.837} C_VEL
LIN {X 0,Y 333.69,Z 227.924,A -85,B 0,C 180,E1 -14348.314,E2 -14348.314} C_VEL
LIN {X 0,Y 333.669,Z 227.927,A -85,B 0,C 180,E1 -14352.506,E2 -14352.506} C_VEL
LIN {X 0,Y 333.67,Z 227.926,A -85,B 0,C 180,E1 -14355.967,E2 -14355.967} C_VEL
LIN {X 0,Y 333.694,Z 227.919,A -85,B 0,C 180,E1 -14359.303,E2 -14359.303} C_VEL
LIN {X 0,Y 333.654,Z 227.919,A -85,B 0,C 180,E1 -14363.167,E2 -14363.167} C_VEL
LIN {X 0,Y 333.624,Z 227.926,A -85,B 0,C 180,E1 -14366.79,E2 -14366.79} C_VEL
LIN {X 0,Y 333.69,Z 227.915,A -85,B 0,C 180,E1 -14369.709,E2 -14369.709} C_VEL
LIN {X 0,Y 333.728,Z 227.907,A -85,B 0,C 180,E1 -14372.4,E2 -14372.4} C_VEL
LIN {X 0,Y 333.709,Z 227.916,A -85,B 0,C 180,E1 -14375.089,E2 -14375.089} C_VEL
LIN {X 0,Y 333.639,Z 227.924,A -85,B 0,C 180,E1 -14379.016,E2 -14379.016} C_VEL
LIN {X 0,Y 333.759,Z 227.907,A -85,B 0,C 180,E1 -14381.587,E2 -14381.587} C_VEL
LIN {X 0,Y 333.79,Z 227.902,A -85,B 0,C 180,E1 -14385.576,E2 -14385.576} C_VEL
LIN {X 0,Y 333.803,Z 227.898,A -85,B 0,C 180,E1 -14389.077,E2 -14389.077} C_VEL
LIN {X 0,Y 333.986,Z 227.88,A -85,B 0,C 180,E1 -14392.747,E2 -14392.747} C_VEL
LIN {X 0,Y 333.782,Z 227.905,A -85,B 0,C 180,E1 -14395.169,E2 -14395.169} C_VEL
LIN {X 0,Y 334.079,Z 227.862,A -85,B 0,C 180,E1 -14397.588,E2 -14397.588} C_VEL
LIN {X 0,Y 334.184,Z 227.855,A -85,B 0,C 180,E1 -14400,E2 -14400} C_VEL
LIN {X 0,Y 334.077,Z 227.865,A -85,B 0,C 180,E1 -14402.411,E2 -14402.411} C_VEL
LIN {X 0,Y 333.973,Z 227.88,A -85,B 0,C 180,E1 -14406.04,E2 -14406.04} C_VEL
LIN {X 0,Y 333.799,Z 227.903,A -85,B 0,C 180,E1 -14409.697,E2 -14409.697} C_VEL
LIN {X 0,Y 333.773,Z 227.905,A -85,B 0,C 180,E1 -14413.392,E2 -14413.392} C_VEL
LIN {X 0,Y 333.737,Z 227.908,A -85,B 0,C 180,E1 -14415.888,E2 -14415.888} C_VEL
LIN {X 0,Y 333.701,Z 227.916,A -85,B 0,C 180,E1 -14418.616,E2 -14418.616} C_VEL
LIN {X 0,Y 333.632,Z 227.919,A -85,B 0,C 180,E1 -14422.282,E2 -14422.282} C_VEL
LIN {X 0,Y 333.643,Z 227.917,A -85,B 0,C 180,E1 -14425.08,E2 -14425.08} C_VEL
LIN {X 0,Y 333.636,Z 227.925,A -85,B 0,C 180,E1 -14427.788,E2 -14427.788} C_VEL
LIN {X 0,Y 333.634,Z 227.92,A -85,B 0,C 180,E1 -14430.369,E2 -14430.369} C_VEL
LIN {X 0,Y 333.619,Z 227.92,A -85,B 0,C 180,E1 -14433.21,E2 -14433.21} C_VEL
LIN {X 0,Y 333.66,Z 227.921,A -85,B 0,C 180,E1 -14436.141,E2 -14436.141} C_VEL
LIN {X 0,Y 333.622,Z 227.907,A -85,B 0,C 180,E1 -14439.196,E2 -14439.196} C_VEL
LIN {X 0,Y 333.622,Z 227.925,A -85,B 0,C 180,E1 -14442.501,E2 -14442.501} C_VEL
LIN {X 0,Y 333.587,Z 227.931,A -85,B 0,C 180,E1 -14445.956,E2 -14445.956} C_VEL
LIN {X 0,Y 333.596,Z 227.927,A -85,B 0,C 180,E1 -14449.326,E2 -14449.326} C_VEL
LIN {X 0,Y 333.658,Z 227.926,A -85,B 0,C 180,E1 -14453.17,E2 -14453.17} C_VEL
LIN {X 0,Y 333.679,Z 228.076,A -85,B 0,C 180,E1 -14455.891,E2 -14455.891} C_VEL
LIN {X 0,Y 336.229,Z 238.417,A -85,B 0,C 180,E1 -14458.981,E2 -14458.981} C_VEL
LIN {X 0,Y 338.546,Z 248.443,A -85,B 0,C 180,E1 -14461.818,E2 -14461.818} C_VEL
LIN {X 0,Y 339.466,Z 253.532,A -85,B 0,C 180,E1 -14463.192,E2 -14463.192} C_VEL
LIN {X 0,Y 338.816,Z 259.47,A -85,B 0,C 180,E1 -14464.626,E2 -14464.626} C_VEL
LIN {X 0,Y 344.437,Z 287.499,A -85,B 0,C 180,E1 -14465.794,E2 -14465.794} C_VEL
LIN {X 0,Y 346.549,Z 301.84,A -85,B 0,C 180,E1 -14466.305,E2 -14466.305} C_VEL
LIN {X 0,Y 344.947,Z 368.841,A -85,B 0,C 180,E1 -14467.739,E2 -14467.739} C_VEL
LIN {X 0,Y 343.985,Z 382.656,A -85,B 0,C 180,E1 -14468.265,E2 -14468.265} C_VEL
LIN {X 0,Y 342.834,Z 395.052,A -85,B 0,C 180,E1 -14468.977,E2 -14468.977} C_VEL
LIN {X 0,Y 341.404,Z 406.148,A -85,B 0,C 180,E1 -14469.83,E2 -14469.83} C_VEL
LIN {X 0,Y 339.768,Z 417.697,A -85,B 0,C 180,E1 -14470.986,E2 -14470.986} C_VEL
LIN {X 0,Y 338.231,Z 428.109,A -85,B 0,C 180,E1 -14472.308,E2 -14472.308} C_VEL
LIN {X 0,Y 336.624,Z 437.706,A -85,B 0,C 180,E1 -14473.819,E2 -14473.819} C_VEL
LIN {X 0,Y 335.393,Z 445.938,A -85,B 0,C 180,E1 -14475.436,E2 -14475.436} C_VEL
LIN {X 0,Y 334.113,Z 453.412,A -85,B 0,C 180,E1 -14477.239,E2 -14477.239} C_VEL
LIN {X 0,Y 333.179,Z 459.446,A -85,B 0,C 180,E1 -14479.055,E2 -14479.055} C_VEL
LIN {X 0,Y 332.567,Z 464.243,A -85,B 0,C 180,E1 -14480.879,E2 -14480.879} C_VEL
LIN {X 0,Y 332.194,Z 467.942,A -85,B 0,C 180,E1 -14482.706,E2 -14482.706} C_VEL
LIN {X 0,Y 332.034,Z 470.198,A -85,B 0,C 180,E1 -14484.17,E2 -14484.17} C_VEL
LIN {X 0,Y 332.012,Z 472.406,A -85,B 0,C 180,E1 -14486.357,E2 -14486.357} C_VEL
LIN {X 0,Y 332.062,Z 473.361,A -85,B 0,C 180,E1 -14488.785,E2 -14488.785} C_VEL
LIN {X 0,Y 332.135,Z 473.236,A -85,B 0,C 180,E1 -14489.998,E2 -14489.998} C_VEL
LIN {X 0,Y 332.104,Z 472.68,A -85,B 0,C 180,E1 -14491.21,E2 -14491.21} C_VEL
LIN {X 0,Y 332.044,Z 470.378,A -85,B 0,C 180,E1 -14493.638,E2 -14493.638} C_VEL
LIN {X 0,Y 332.062,Z 468.58,A -85,B 0,C 180,E1 -14494.854,E2 -14494.854} C_VEL
LIN {X 0,Y 332.155,Z 465.02,A -85,B 0,C 180,E1 -14496.68,E2 -14496.68} C_VEL
LIN {X 0,Y 332.35,Z 460.33,A -85,B 0,C 180,E1 -14498.509,E2 -14498.509} C_VEL
LIN {X 0,Y 332.821,Z 453.237,A -85,B 0,C 180,E1 -14500.644,E2 -14500.644} C_VEL
LIN {X 0,Y 333.608,Z 445.561,A -85,B 0,C 180,E1 -14502.467,E2 -14502.467} C_VEL
LIN {X 0,Y 334.415,Z 437.689,A -85,B 0,C 180,E1 -14503.982,E2 -14503.982} C_VEL
LIN {X 0,Y 335.248,Z 429.088,A -85,B 0,C 180,E1 -14505.35,E2 -14505.35} C_VEL
LIN {X 0,Y 336.293,Z 418.664,A -85,B 0,C 180,E1 -14506.696,E2 -14506.696} C_VEL
LIN {X 0,Y 337.449,Z 407.048,A -85,B 0,C 180,E1 -14507.886,E2 -14507.886} C_VEL
LIN {X 0,Y 338.477,Z 394.798,A -85,B 0,C 180,E1 -14508.848,E2 -14508.848} C_VEL
LIN {X 0,Y 339.459,Z 381.152,A -85,B 0,C 180,E1 -14509.616,E2 -14509.616} C_VEL
LIN {X 0,Y 340.076,Z 368.364,A -85,B 0,C 180,E1 -14510.09,E2 -14510.09} C_VEL
LIN {X 0,Y 341.181,Z 298.849,A -85,B 0,C 180,E1 -14511.566,E2 -14511.566} C_VEL
LIN {X 0,Y 336.036,Z 260.177,A -85,B 0,C 180,E1 -14512.717,E2 -14512.717} C_VEL
LIN {X 0,Y 337.259,Z 247.682,A -85,B 0,C 180,E1 -14515.615,E2 -14515.615} C_VEL
LIN {X 0,Y 336.829,Z 243.084,A -85,B 0,C 180,E1 -14516.742,E2 -14516.742} C_VEL
LIN {X 0,Y 334.281,Z 230.635,A -85,B 0,C 180,E1 -14519.949,E2 -14519.949} C_VEL
LIN {X 0,Y 333.686,Z 227.922,A -85,B 0,C 180,E1 -14520.707,E2 -14520.707} C_VEL
LIN {X 0,Y 333.667,Z 227.92,A -85,B 0,C 180,E1 -14524.769,E2 -14524.769} C_VEL
LIN {X 0,Y 333.631,Z 227.927,A -85,B 0,C 180,E1 -14527.647,E2 -14527.647} C_VEL
LIN {X 0,Y 333.624,Z 227.925,A -85,B 0,C 180,E1 -14530.763,E2 -14530.763} C_VEL
LIN {X 0,Y 333.605,Z 227.929,A -85,B 0,C 180,E1 -14534.252,E2 -14534.252} C_VEL
LIN {X 0,Y 333.667,Z 227.923,A -85,B 0,C 180,E1 -14537.622,E2 -14537.622} C_VEL
LIN {X 0,Y 333.648,Z 227.923,A -85,B 0,C 180,E1 -14541.192,E2 -14541.192} C_VEL
LIN {X 0,Y 333.651,Z 227.923,A -85,B 0,C 180,E1 -14545.222,E2 -14545.222} C_VEL
LIN {X 0,Y 333.661,Z 227.925,A -85,B 0,C 180,E1 -14549.634,E2 -14549.634} C_VEL
LIN {X 0,Y 333.704,Z 227.914,A -85,B 0,C 180,E1 -14552.398,E2 -14552.398} C_VEL
LIN {X 0,Y 333.685,Z 227.917,A -85,B 0,C 180,E1 -14556.411,E2 -14556.411} C_VEL
LIN {X 0,Y 333.715,Z 227.913,A -85,B 0,C 180,E1 -14560.308,E2 -14560.308} C_VEL
LIN {X 0,Y 333.733,Z 227.911,A -85,B 0,C 180,E1 -14564.112,E2 -14564.112} C_VEL
LIN {X 0,Y 333.748,Z 227.91,A -85,B 0,C 180,E1 -14567.844,E2 -14567.844} C_VEL
LIN {X 0,Y 333.934,Z 227.888,A -85,B 0,C 180,E1 -14571.528,E2 -14571.528} C_VEL
LIN {X 0,Y 333.978,Z 227.88,A -85,B 0,C 180,E1 -14573.96,E2 -14573.96} C_VEL
LIN {X 0,Y 334.059,Z 227.871,A -85,B 0,C 180,E1 -14577.589,E2 -14577.589} C_VEL
LIN {X 0,Y 334.178,Z 227.854,A -85,B 0,C 180,E1 -14580,E2 -14580} C_VEL
LIN {X 0,Y 334.054,Z 227.868,A -85,B 0,C 180,E1 -14582.412,E2 -14582.412} C_VEL
LIN {X 0,Y 333.942,Z 227.883,A -85,B 0,C 180,E1 -14586.705,E2 -14586.705} C_VEL
LIN {X 0,Y 333.805,Z 227.901,A -85,B 0,C 180,E1 -14589.697,E2 -14589.697} C_VEL
LIN {X 0,Y 333.749,Z 227.907,A -85,B 0,C 180,E1 -14593.394,E2 -14593.394} C_VEL
LIN {X 0,Y 333.685,Z 227.918,A -85,B 0,C 180,E1 -14597.15,E2 -14597.15} C_VEL
LIN {X 0,Y 333.62,Z 227.925,A -85,B 0,C 180,E1 -14599.698,E2 -14599.698} C_VEL
LIN {X 0,Y 333.627,Z 227.923,A -85,B 0,C 180,E1 -14603.594,E2 -14603.594} C_VEL
LIN {X 0,Y 333.696,Z 227.918,A -85,B 0,C 180,E1 -14606.25,E2 -14606.25} C_VEL
LIN {X 0,Y 333.674,Z 227.919,A -85,B 0,C 180,E1 -14608.976,E2 -14608.976} C_VEL
LIN {X 0,Y 333.608,Z 227.931,A -85,B 0,C 180,E1 -14612.59,E2 -14612.59} C_VEL
LIN {X 0,Y 333.643,Z 227.925,A -85,B 0,C 180,E1 -14616.143,E2 -14616.143} C_VEL
LIN {X 0,Y 333.652,Z 227.92,A -85,B 0,C 180,E1 -14619.192,E2 -14619.192} C_VEL
LIN {X 0,Y 333.663,Z 227.923,A -85,B 0,C 180,E1 -14622.515,E2 -14622.515} C_VEL
LIN {X 0,Y 333.601,Z 227.929,A -85,B 0,C 180,E1 -14625.964,E2 -14625.964} C_VEL
LIN {X 0,Y 333.625,Z 227.924,A -85,B 0,C 180,E1 -14629.32,E2 -14629.32} C_VEL
LIN {X 0,Y 333.646,Z 227.92,A -85,B 0,C 180,E1 -14633.173,E2 -14633.173} C_VEL
LIN {X 0,Y 333.657,Z 227.92,A -85,B 0,C 180,E1 -14635.346,E2 -14635.346} C_VEL
LIN {X 0,Y 333.677,Z 227.92,A -85,B 0,C 180,E1 -14639.642,E2 -14639.642} C_VEL
LIN {X 0,Y 333.728,Z 227.913,A -85,B 0,C 180,E1 -14642.405,E2 -14642.405} C_VEL
LIN {X 0,Y 333.716,Z 227.913,A -85,B 0,C 180,E1 -14645.095,E2 -14645.095} C_VEL
LIN {X 0,Y 333.663,Z 227.919,A -85,B 0,C 180,E1 -14649.023,E2 -14649.023} C_VEL
LIN {X 0,Y 333.736,Z 227.914,A -85,B 0,C 180,E1 -14651.59,E2 -14651.59} C_VEL
LIN {X 0,Y 333.806,Z 227.907,A -85,B 0,C 180,E1 -14655.58,E2 -14655.58} C_VEL
LIN {X 0,Y 333.827,Z 228.049,A -85,B 0,C 180,E1 -14657.233,E2 -14657.233} C_VEL
LIN {X 0,Y 334.566,Z 231.773,A -85,B 0,C 180,E1 -14658.288,E2 -14658.288} C_VEL
LIN {X 0,Y 340.222,Z 249.021,A -85,B 0,C 180,E1 -14659.011,E2 -14659.011} C_VEL
LIN {X 0,Y 341.916,Z 258.748,A -85,B 0,C 180,E1 -14659.32,E2 -14659.32} C_VEL
LIN {X 0,Y 340.273,Z 339.295,A -85,B 0,C 180,E1 -14661.017,E2 -14661.017} C_VEL
LIN {X 0,Y 339.716,Z 352.404,A -85,B 0,C 180,E1 -14661.527,E2 -14661.527} C_VEL
LIN {X 0,Y 339.109,Z 363.876,A -85,B 0,C 180,E1 -14662.186,E2 -14662.186} C_VEL
LIN {X 0,Y 338.516,Z 374.461,A -85,B 0,C 180,E1 -14662.997,E2 -14662.997} C_VEL
LIN {X 0,Y 337.508,Z 385.19,A -85,B 0,C 180,E1 -14664.027,E2 -14664.027} C_VEL
LIN {X 0,Y 336.545,Z 395.045,A -85,B 0,C 180,E1 -14665.211,E2 -14665.211} C_VEL
LIN {X 0,Y 335.487,Z 405,A -85,B 0,C 180,E1 -14666.7,E2 -14666.7} C_VEL
LIN {X 0,Y 334.526,Z 414.624,A -85,B 0,C 180,E1 -14668.498,E2 -14668.498} C_VEL
LIN {X 0,Y 333.624,Z 422.332,A -85,B 0,C 180,E1 -14670.304,E2 -14670.304} C_VEL
LIN {X 0,Y 333.028,Z 429.395,A -85,B 0,C 180,E1 -14672.421,E2 -14672.421} C_VEL
LIN {X 0,Y 332.562,Z 434.122,A -85,B 0,C 180,E1 -14674.244,E2 -14674.244} C_VEL
LIN {X 0,Y 332.332,Z 438.154,A -85,B 0,C 180,E1 -14676.311,E2 -14676.311} C_VEL
LIN {X 0,Y 332.056,Z 441.016,A -85,B 0,C 180,E1 -14678.522,E2 -14678.522} C_VEL
LIN {X 0,Y 331.976,Z 442.635,A -85,B 0,C 180,E1 -14680.985,E2 -14680.985} C_VEL
LIN {X 0,Y 332.115,Z 442.696,A -85,B 0,C 180,E1 -14683.238,E2 -14683.238} C_VEL
LIN {X 0,Y 332.251,Z 441.99,A -85,B 0,C 180,E1 -14684.705,E2 -14684.705} C_VEL
LIN {X 0,Y 332.414,Z 440.97,A -85,B 0,C 180,E1 -14685.954,E2 -14685.954} C_VEL
LIN {X 0,Y 333.016,Z 437.901,A -85,B 0,C 180,E1 -14688.251,E2 -14688.251} C_VEL
LIN {X 0,Y 333.767,Z 433.773,A -85,B 0,C 180,E1 -14690.331,E2 -14690.331} C_VEL
LIN {X 0,Y 334.672,Z 428.799,A -85,B 0,C 180,E1 -14692.21,E2 -14692.21} C_VEL
LIN {X 0,Y 335.829,Z 422.474,A -85,B 0,C 180,E1 -14694.084,E2 -14694.084} C_VEL
LIN {X 0,Y 337.011,Z 415.947,A -85,B 0,C 180,E1 -14695.64,E2 -14695.64} C_VEL
LIN {X 0,Y 338.355,Z 408.044,A -85,B 0,C 180,E1 -14697.191,E2 -14697.191} C_VEL
LIN {X 0,Y 339.859,Z 398.283,A -85,B 0,C 180,E1 -14698.736,E2 -14698.736} C_VEL
LIN {X 0,Y 341.415,Z 387.984,A -85,B 0,C 180,E1 -14700.038,E2 -14700.038} C_VEL
LIN {X 0,Y 342.817,Z 376.737,A -85,B 0,C 180,E1 -14701.173,E2 -14701.173} C_VEL
LIN {X 0,Y 343.851,Z 364.927,A -85,B 0,C 180,E1 -14702.1,E2 -14702.1} C_VEL
LIN {X 0,Y 344.915,Z 351.488,A -85,B 0,C 180,E1 -14702.854,E2 -14702.854} C_VEL
LIN {X 0,Y 345.516,Z 339.309,A -85,B 0,C 180,E1 -14703.311,E2 -14703.311} C_VEL
LIN {X 0,Y 346.317,Z 305.185,A -85,B 0,C 180,E1 -14704.051,E2 -14704.051} C_VEL
LIN {X 0,Y 345.891,Z 299.386,A -85,B 0,C 180,E1 -14704.22,E2 -14704.22} C_VEL
LIN {X 0,Y 341.395,Z 280.722,A -85,B 0,C 180,E1 -14705.046,E2 -14705.046} C_VEL
LIN {X 0,Y 340.904,Z 274.925,A -85,B 0,C 180,E1 -14705.227,E2 -14705.227} C_VEL
LIN {X 0,Y 341.123,Z 262.37,A -85,B 0,C 180,E1 -14705.503,E2 -14705.503} C_VEL
LIN {X 0,Y 332.724,Z 243.263,A -85,B 0,C 180,E1 -14706.763,E2 -14706.763} C_VEL
LIN {X 0,Y 327.656,Z 232.842,A -85,B 0,C 180,E1 -14707.567,E2 -14707.567} C_VEL
LIN {X 0,Y 326.646,Z 228.804,A -85,B 0,C 180,E1 -14708.915,E2 -14708.915} C_VEL
LIN {X 0,Y 326.61,Z 228.8,A -85,B 0,C 180,E1 -14712.978,E2 -14712.978} C_VEL
LIN {X 0,Y 326.622,Z 228.8,A -85,B 0,C 180,E1 -14717.017,E2 -14717.017} C_VEL
LIN {X 0,Y 326.634,Z 228.798,A -85,B 0,C 180,E1 -14720.765,E2 -14720.765} C_VEL
LIN {X 0,Y 326.601,Z 228.801,A -85,B 0,C 180,E1 -14724.479,E2 -14724.479} C_VEL
LIN {X 0,Y 326.595,Z 228.804,A -85,B 0,C 180,E1 -14727.454,E2 -14727.454} C_VEL
LIN {X 0,Y 326.647,Z 228.797,A -85,B 0,C 180,E1 -14730.339,E2 -14730.339} C_VEL
LIN {X 0,Y 326.675,Z 228.792,A -85,B 0,C 180,E1 -14734.515,E2 -14734.515} C_VEL
LIN {X 0,Y 326.594,Z 228.801,A -85,B 0,C 180,E1 -14738.541,E2 -14738.541} C_VEL
LIN {X 0,Y 326.692,Z 228.783,A -85,B 0,C 180,E1 -14741.174,E2 -14741.174} C_VEL
LIN {X 0,Y 326.745,Z 228.778,A -85,B 0,C 180,E1 -14745.433,E2 -14745.433} C_VEL
LIN {X 0,Y 326.742,Z 228.777,A -85,B 0,C 180,E1 -14748.838,E2 -14748.838} C_VEL
LIN {X 0,Y 326.936,Z 228.758,A -85,B 0,C 180,E1 -14752.589,E2 -14752.589} C_VEL
LIN {X 0,Y 326.967,Z 228.749,A -85,B 0,C 180,E1 -14753.83,E2 -14753.83} C_VEL
LIN {X 0,Y 327.02,Z 228.742,A -85,B 0,C 180,E1 -14757.536,E2 -14757.536} C_VEL
LIN {X 0,Y 327.137,Z 228.733,A -85,B 0,C 180,E1 -14760,E2 -14760} C_VEL
LIN {X 0,Y 327.018,Z 228.744,A -85,B 0,C 180,E1 -14762.463,E2 -14762.463} C_VEL
LIN {X 0,Y 326.927,Z 228.758,A -85,B 0,C 180,E1 -14766.17,E2 -14766.17} C_VEL
LIN {X 0,Y 326.763,Z 228.78,A -85,B 0,C 180,E1 -14769.908,E2 -14769.908} C_VEL
LIN {X 0,Y 326.737,Z 228.782,A -85,B 0,C 180,E1 -14773.686,E2 -14773.686} C_VEL
LIN {X 0,Y 326.643,Z 228.79,A -85,B 0,C 180,E1 -14777.531,E2 -14777.531} C_VEL
LIN {X 0,Y 326.592,Z 228.794,A -85,B 0,C 180,E1 -14781.458,E2 -14781.458} C_VEL
LIN {X 0,Y 326.586,Z 228.794,A -85,B 0,C 180,E1 -14785.492,E2 -14785.492} C_VEL
LIN {X 0,Y 326.578,Z 228.806,A -85,B 0,C 180,E1 -14788.258,E2 -14788.258} C_VEL
LIN {X 0,Y 326.55,Z 228.808,A -85,B 0,C 180,E1 -14791.1,E2 -14791.1} C_VEL
LIN {X 0,Y 326.591,Z 228.796,A -85,B 0,C 180,E1 -14794.021,E2 -14794.021} C_VEL
LIN {X 0,Y 326.61,Z 228.787,A -85,B 0,C 180,E1 -14797.238,E2 -14797.238} C_VEL
LIN {X 0,Y 326.566,Z 228.806,A -85,B 0,C 180,E1 -14801.132,E2 -14801.132} C_VEL
LIN {X 0,Y 326.518,Z 228.81,A -85,B 0,C 180,E1 -14804.744,E2 -14804.744} C_VEL
LIN {X 0,Y 326.556,Z 228.797,A -85,B 0,C 180,E1 -14808.153,E2 -14808.153} C_VEL
LIN {X 0,Y 326.562,Z 228.8,A -85,B 0,C 180,E1 -14811.384,E2 -14811.384} C_VEL
LIN {X 0,Y 326.659,Z 228.791,A -85,B 0,C 180,E1 -14815.171,E2 -14815.171} C_VEL
LIN {X 0,Y 329.098,Z 238.66,A -85,B 0,C 180,E1 -14818.283,E2 -14818.283} C_VEL
LIN {X 0,Y 331.647,Z 249.794,A -85,B 0,C 180,E1 -14821.524,E2 -14821.524} C_VEL
LIN {X 0,Y 332.639,Z 255.76,A -85,B 0,C 180,E1 -14823.163,E2 -14823.163} C_VEL
LIN {X 0,Y 332.21,Z 259.083,A -85,B 0,C 180,E1 -14823.978,E2 -14823.978} C_VEL
LIN {X 0,Y 337.498,Z 284.956,A -85,B 0,C 180,E1 -14825.115,E2 -14825.115} C_VEL
LIN {X 0,Y 340.23,Z 302.372,A -85,B 0,C 180,E1 -14825.772,E2 -14825.772} C_VEL
LIN {X 0,Y 338.571,Z 368.588,A -85,B 0,C 180,E1 -14827.216,E2 -14827.216} C_VEL
LIN {X 0,Y 337.581,Z 382.376,A -85,B 0,C 180,E1 -14827.75,E2 -14827.75} C_VEL
LIN {X 0,Y 336.387,Z 394.757,A -85,B 0,C 180,E1 -14828.474,E2 -14828.474} C_VEL
LIN {X 0,Y 334.784,Z 406.631,A -85,B 0,C 180,E1 -14829.413,E2 -14829.413} C_VEL
LIN {X 0,Y 333.08,Z 418.032,A -85,B 0,C 180,E1 -14830.59,E2 -14830.59} C_VEL
LIN {X 0,Y 331.485,Z 428.331,A -85,B 0,C 180,E1 -14831.936,E2 -14831.936} C_VEL
LIN {X 0,Y 329.927,Z 437.121,A -85,B 0,C 180,E1 -14833.35,E2 -14833.35} C_VEL
LIN {X 0,Y 328.499,Z 445.957,A -85,B 0,C 180,E1 -14835.123,E2 -14835.123} C_VEL
LIN {X 0,Y 327.189,Z 453.37,A -85,B 0,C 180,E1 -14836.964,E2 -14836.964} C_VEL
LIN {X 0,Y 326.161,Z 459.346,A -85,B 0,C 180,E1 -14838.817,E2 -14838.817} C_VEL
LIN {X 0,Y 325.543,Z 464.093,A -85,B 0,C 180,E1 -14840.681,E2 -14840.681} C_VEL
LIN {X 0,Y 325.144,Z 467.745,A -85,B 0,C 180,E1 -14842.547,E2 -14842.547} C_VEL
LIN {X 0,Y 324.93,Z 470.193,A -85,B 0,C 180,E1 -14844.239,E2 -14844.239} C_VEL
LIN {X 0,Y 324.937,Z 472.127,A -85,B 0,C 180,E1 -14846.278,E2 -14846.278} C_VEL
LIN {X 0,Y 324.964,Z 473.042,A -85,B 0,C 180,E1 -14848.759,E2 -14848.759} C_VEL
LIN {X 0,Y 325.043,Z 472.88,A -85,B 0,C 180,E1 -14849.998,E2 -14849.998} C_VEL
LIN {X 0,Y 325.007,Z 472.303,A -85,B 0,C 180,E1 -14851.237,E2 -14851.237} C_VEL
LIN {X 0,Y 324.971,Z 469.962,A -85,B 0,C 180,E1 -14853.717,E2 -14853.717} C_VEL
LIN {X 0,Y 325.003,Z 466.464,A -85,B 0,C 180,E1 -14855.887,E2 -14855.887} C_VEL
LIN {X 0,Y 325.213,Z 461.479,A -85,B 0,C 180,E1 -14858.072,E2 -14858.072} C_VEL
LIN {X 0,Y 325.568,Z 455.922,A -85,B 0,C 180,E1 -14859.941,E2 -14859.941} C_VEL
LIN {X 0,Y 326.155,Z 448.969,A -85,B 0,C 180,E1 -14861.809,E2 -14861.809} C_VEL
LIN {X 0,Y 326.948,Z 441.868,A -85,B 0,C 180,E1 -14863.357,E2 -14863.357} C_VEL
LIN {X 0,Y 327.843,Z 433.286,A -85,B 0,C 180,E1 -14864.903,E2 -14864.903} C_VEL
LIN {X 0,Y 328.942,Z 422.66,A -85,B 0,C 180,E1 -14866.441,E2 -14866.441} C_VEL
LIN {X 0,Y 330.007,Z 412.134,A -85,B 0,C 180,E1 -14867.662,E2 -14867.662} C_VEL
LIN {X 0,Y 331.137,Z 400.564,A -85,B 0,C 180,E1 -14868.72,E2 -14868.72} C_VEL
LIN {X 0,Y 332.097,Z 388.55,A -85,B 0,C 180,E1 -14869.546,E2 -14869.546} C_VEL
LIN {X 0,Y 332.922,Z 375.565,A -85,B 0,C 180,E1 -14870.178,E2 -14870.178} C_VEL
LIN {X 0,Y 333.424,Z 363.446,A -85,B 0,C 180,E1 -14870.549,E2 -14870.549} C_VEL
LIN {X 0,Y 334.404,Z 299.728,A -85,B 0,C 180,E1 -14871.914,E2 -14871.914} C_VEL
LIN {X 0,Y 329.177,Z 259.83,A -85,B 0,C 180,E1 -14873.136,E2 -14873.136} C_VEL
LIN {X 0,Y 330.318,Z 248.357,A -85,B 0,C 180,E1 -14875.854,E2 -14875.854} C_VEL
LIN {X 0,Y 329.524,Z 242.71,A -85,B 0,C 180,E1 -14877.287,E2 -14877.287} C_VEL
LIN {X 0,Y 327.245,Z 231.598,A -85,B 0,C 180,E1 -14880.224,E2 -14880.224} C_VEL
LIN {X 0,Y 326.616,Z 228.804,A -85,B 0,C 180,E1 -14881.015,E2 -14881.015} C_VEL
LIN {X 0,Y 326.589,Z 228.807,A -85,B 0,C 180,E1 -14884.015,E2 -14884.015} C_VEL
LIN {X 0,Y 326.607,Z 228.8,A -85,B 0,C 180,E1 -14887.234,E2 -14887.234} C_VEL
LIN {X 0,Y 326.555,Z 228.805,A -85,B 0,C 180,E1 -14891.126,E2 -14891.126} C_VEL
LIN {X 0,Y 326.544,Z 228.806,A -85,B 0,C 180,E1 -14894.746,E2 -14894.746} C_VEL
LIN {X 0,Y 326.594,Z 228.803,A -85,B 0,C 180,E1 -14898.157,E2 -14898.157} C_VEL
LIN {X 0,Y 326.613,Z 228.8,A -85,B 0,C 180,E1 -14901.39,E2 -14901.39} C_VEL
LIN {X 0,Y 326.585,Z 228.802,A -85,B 0,C 180,E1 -14904.848,E2 -14904.848} C_VEL
LIN {X 0,Y 326.572,Z 228.807,A -85,B 0,C 180,E1 -14907.452,E2 -14907.452} C_VEL
LIN {X 0,Y 326.624,Z 228.797,A -85,B 0,C 180,E1 -14910.337,E2 -14910.337} C_VEL
LIN {X 0,Y 326.655,Z 228.792,A -85,B 0,C 180,E1 -14914.513,E2 -14914.513} C_VEL
LIN {X 0,Y 326.638,Z 228.794,A -85,B 0,C 180,E1 -14918.545,E2 -14918.545} C_VEL
LIN {X 0,Y 326.704,Z 228.79,A -85,B 0,C 180,E1 -14921.175,E2 -14921.175} C_VEL
LIN {X 0,Y 326.72,Z 228.788,A -85,B 0,C 180,E1 -14925.432,E2 -14925.432} C_VEL
LIN {X 0,Y 326.727,Z 228.785,A -85,B 0,C 180,E1 -14928.838,E2 -14928.838} C_VEL
LIN {X 0,Y 326.934,Z 228.758,A -85,B 0,C 180,E1 -14932.589,E2 -14932.589} C_VEL
LIN {X 0,Y 326.735,Z 228.787,A -85,B 0,C 180,E1 -14935.064,E2 -14935.064} C_VEL
LIN {X 0,Y 327,Z 228.75,A -85,B 0,C 180,E1 -14937.537,E2 -14937.537} C_VEL
LIN {X 0,Y 327.13,Z 228.731,A -85,B 0,C 180,E1 -14940,E2 -14940} C_VEL
LIN {X 0,Y 326.995,Z 228.746,A -85,B 0,C 180,E1 -14942.464,E2 -14942.464} C_VEL
LIN {X 0,Y 326.907,Z 228.759,A -85,B 0,C 180,E1 -14946.697,E2 -14946.697} C_VEL
LIN {X 0,Y 326.761,Z 228.779,A -85,B 0,C 180,E1 -14949.908,E2 -14949.908} C_VEL
LIN {X 0,Y 326.713,Z 228.781,A -85,B 0,C 180,E1 -14953.688,E2 -14953.688} C_VEL
LIN {X 0,Y 326.631,Z 228.795,A -85,B 0,C 180,E1 -14957.532,E2 -14957.532} C_VEL
LIN {X 0,Y 326.569,Z 228.803,A -85,B 0,C 180,E1 -14961.46,E2 -14961.46} C_VEL
LIN {X 0,Y 326.651,Z 228.793,A -85,B 0,C 180,E1 -14965.487,E2 -14965.487} C_VEL
LIN {X 0,Y 326.624,Z 228.796,A -85,B 0,C 180,E1 -14969.663,E2 -14969.663} C_VEL
LIN {X 0,Y 326.573,Z 228.804,A -85,B 0,C 180,E1 -14974.024,E2 -14974.024} C_VEL
LIN {X 0,Y 326.596,Z 228.8,A -85,B 0,C 180,E1 -14977.242,E2 -14977.242} C_VEL
LIN {X 0,Y 326.606,Z 228.802,A -85,B 0,C 180,E1 -14980.207,E2 -14980.207} C_VEL
LIN {X 0,Y 326.588,Z 228.8,A -85,B 0,C 180,E1 -14983.522,E2 -14983.522} C_VEL
LIN {X 0,Y 326.56,Z 228.803,A -85,B 0,C 180,E1 -14987.032,E2 -14987.032} C_VEL
LIN {X 0,Y 326.591,Z 228.8,A -85,B 0,C 180,E1 -14990.778,E2 -14990.778} C_VEL
LIN {X 0,Y 326.595,Z 228.802,A -85,B 0,C 180,E1 -14994.485,E2 -14994.485} C_VEL
LIN {X 0,Y 326.593,Z 228.801,A -85,B 0,C 180,E1 -14997.46,E2 -14997.46} C_VEL
LIN {X 0,Y 326.635,Z 228.797,A -85,B 0,C 180,E1 -15000.344,E2 -15000.344} C_VEL
LIN {X 0,Y 326.68,Z 228.79,A -85,B 0,C 180,E1 -15004.521,E2 -15004.521} C_VEL
LIN {X 0,Y 326.611,Z 228.798,A -85,B 0,C 180,E1 -15008.548,E2 -15008.548} C_VEL
LIN {X 0,Y 326.659,Z 228.793,A -85,B 0,C 180,E1 -15012.474,E2 -15012.474} C_VEL
LIN {X 0,Y 326.757,Z 228.782,A -85,B 0,C 180,E1 -15016.318,E2 -15016.318} C_VEL
LIN {X 0,Y 326.799,Z 228.99,A -85,B 0,C 180,E1 -15016.953,E2 -15016.953} C_VEL
LIN {X 0,Y 327.407,Z 232.068,A -85,B 0,C 180,E1 -15017.843,E2 -15017.843} C_VEL
LIN {X 0,Y 333.641,Z 250.684,A -85,B 0,C 180,E1 -15018.665,E2 -15018.665} C_VEL
LIN {X 0,Y 335.087,Z 258.759,A -85,B 0,C 180,E1 -15018.931,E2 -15018.931} C_VEL
LIN {X 0,Y 333.493,Z 338.591,A -85,B 0,C 180,E1 -15020.642,E2 -15020.642} C_VEL
LIN {X 0,Y 332.896,Z 352.104,A -85,B 0,C 180,E1 -15021.161,E2 -15021.161} C_VEL
LIN {X 0,Y 332.271,Z 364.282,A -85,B 0,C 180,E1 -15021.871,E2 -15021.871} C_VEL
LIN {X 0,Y 331.646,Z 374.85,A -85,B 0,C 180,E1 -15022.698,E2 -15022.698} C_VEL
LIN {X 0,Y 330.619,Z 385.564,A -85,B 0,C 180,E1 -15023.749,E2 -15023.749} C_VEL
LIN {X 0,Y 329.62,Z 395.409,A -85,B 0,C 180,E1 -15024.957,E2 -15024.957} C_VEL
LIN {X 0,Y 328.649,Z 404.468,A -85,B 0,C 180,E1 -15026.324,E2 -15026.324} C_VEL
LIN {X 0,Y 327.773,Z 412.762,A -85,B 0,C 180,E1 -15027.852,E2 -15027.852} C_VEL
LIN {X 0,Y 326.831,Z 420.893,A -85,B 0,C 180,E1 -15029.694,E2 -15029.694} C_VEL
LIN {X 0,Y 326.191,Z 426.439,A -85,B 0,C 180,E1 -15031.237,E2 -15031.237} C_VEL
LIN {X 0,Y 325.772,Z 431.843,A -85,B 0,C 180,E1 -15033.094,E2 -15033.094} C_VEL
LIN {X 0,Y 325.426,Z 436.086,A -85,B 0,C 180,E1 -15034.958,E2 -15034.958} C_VEL
LIN {X 0,Y 325.252,Z 438.496,A -85,B 0,C 180,E1 -15036.295,E2 -15036.295} C_VEL
LIN {X 0,Y 325.115,Z 440.134,A -85,B 0,C 180,E1 -15037.454,E2 -15037.454} C_VEL
LIN {X 0,Y 324.96,Z 441.494,A -85,B 0,C 180,E1 -15038.709,E2 -15038.709} C_VEL
LIN {X 0,Y 324.887,Z 443.026,A -85,B 0,C 180,E1 -15041.228,E2 -15041.228} C_VEL
LIN {X 0,Y 325.037,Z 443.033,A -85,B 0,C 180,E1 -15043.344,E2 -15043.344} C_VEL
LIN {X 0,Y 325.211,Z 442.216,A -85,B 0,C 180,E1 -15045.031,E2 -15045.031} C_VEL
LIN {X 0,Y 325.404,Z 441.136,A -85,B 0,C 180,E1 -15046.307,E2 -15046.307} C_VEL
LIN {X 0,Y 326.022,Z 438.266,A -85,B 0,C 180,E1 -15048.467,E2 -15048.467} C_VEL
LIN {X 0,Y 326.884,Z 433.727,A -85,B 0,C 180,E1 -15050.778,E2 -15050.778} C_VEL
LIN {X 0,Y 327.983,Z 428.139,A -85,B 0,C 180,E1 -15052.867,E2 -15052.867} C_VEL
LIN {X 0,Y 329.355,Z 420.927,A -85,B 0,C 180,E1 -15054.925,E2 -15054.925} C_VEL
LIN {X 0,Y 330.681,Z 414.012,A -85,B 0,C 180,E1 -15056.507,E2 -15056.507} C_VEL
LIN {X 0,Y 332.131,Z 405.603,A -85,B 0,C 180,E1 -15058.087,E2 -15058.087} C_VEL
LIN {X 0,Y 333.588,Z 396.365,A -85,B 0,C 180,E1 -15059.502,E2 -15059.502} C_VEL
LIN {X 0,Y 335.298,Z 385.222,A -85,B 0,C 180,E1 -15060.851,E2 -15060.851} C_VEL
LIN {X 0,Y 336.681,Z 373.365,A -85,B 0,C 180,E1 -15061.983,E2 -15061.983} C_VEL
LIN {X 0,Y 337.658,Z 362.835,A -85,B 0,C 180,E1 -15062.762,E2 -15062.762} C_VEL
LIN {X 0,Y 338.659,Z 350.046,A -85,B 0,C 180,E1 -15063.451,E2 -15063.451} C_VEL
LIN {X 0,Y 339.214,Z 337.382,A -85,B 0,C 180,E1 -15063.894,E2 -15063.894} C_VEL
LIN {X 0,Y 340.904,Z 274.925,A -85,B 0,C 180,E1 -15065.227,E2 -15065.227} C_VEL
LIN {X 0,Y 340.504,Z 271.109,A -85,B 0,C 180,E1 -15065.353,E2 -15065.353} C_VEL
LIN {X 0,Y 339.409,Z 267.502,A -85,B 0,C 180,E1 -15065.539,E2 -15065.539} C_VEL
LIN {X 0,Y 336.902,Z 262.494,A -85,B 0,C 180,E1 -15065.893,E2 -15065.893} C_VEL
LIN {X 0,Y 329.563,Z 251.455,A -85,B 0,C 180,E1 -15066.876,E2 -15066.876} C_VEL
LIN {X 0,Y 327.761,Z 248.063,A -85,B 0,C 180,E1 -15067.143,E2 -15067.143} C_VEL
LIN {X 0,Y 320.481,Z 233.307,A -85,B 0,C 180,E1 -15068.3,E2 -15068.3} C_VEL
LIN {X 0,Y 319.576,Z 229.676,A -85,B 0,C 180,E1 -15069.564,E2 -15069.564} C_VEL
LIN {X 0,Y 319.581,Z 229.669,A -85,B 0,C 180,E1 -15073.471,E2 -15073.471} C_VEL
LIN {X 0,Y 319.597,Z 229.674,A -85,B 0,C 180,E1 -15077.023,E2 -15077.023} C_VEL
LIN {X 0,Y 319.575,Z 229.676,A -85,B 0,C 180,E1 -15080.375,E2 -15080.375} C_VEL
LIN {X 0,Y 319.548,Z 229.678,A -85,B 0,C 180,E1 -15083.571,E2 -15083.571} C_VEL
LIN {X 0,Y 319.567,Z 229.678,A -85,B 0,C 180,E1 -15086.685,E2 -15086.685} C_VEL
LIN {X 0,Y 319.579,Z 229.672,A -85,B 0,C 180,E1 -15089.615,E2 -15089.615} C_VEL
LIN {X 0,Y 319.594,Z 229.667,A -85,B 0,C 180,E1 -15092.496,E2 -15092.496} C_VEL
LIN {X 0,Y 319.588,Z 229.675,A -85,B 0,C 180,E1 -15095.302,E2 -15095.302} C_VEL
LIN {X 0,Y 319.564,Z 229.676,A -85,B 0,C 180,E1 -15099.397,E2 -15099.397} C_VEL
LIN {X 0,Y 319.625,Z 229.671,A -85,B 0,C 180,E1 -15102.071,E2 -15102.071} C_VEL
LIN {X 0,Y 319.712,Z 229.66,A -85,B 0,C 180,E1 -15106.007,E2 -15106.007} C_VEL
LIN {X 0,Y 319.721,Z 229.655,A -85,B 0,C 180,E1 -15109.871,E2 -15109.871} C_VEL
LIN {X 0,Y 319.922,Z 229.626,A -85,B 0,C 180,E1 -15113.694,E2 -15113.694} C_VEL
LIN {X 0,Y 319.964,Z 229.621,A -85,B 0,C 180,E1 -15117.482,E2 -15117.482} C_VEL
LIN {X 0,Y 320.09,Z 229.611,A -85,B 0,C 180,E1 -15120,E2 -15120} C_VEL
LIN {X 0,Y 319.962,Z 229.622,A -85,B 0,C 180,E1 -15122.518,E2 -15122.518} C_VEL
LIN {X 0,Y 319.884,Z 229.636,A -85,B 0,C 180,E1 -15126.307,E2 -15126.307} C_VEL
LIN {X 0,Y 319.715,Z 229.658,A -85,B 0,C 180,E1 -15130.128,E2 -15130.128} C_VEL
LIN {X 0,Y 319.712,Z 229.657,A -85,B 0,C 180,E1 -15133.993,E2 -15133.993} C_VEL
LIN {X 0,Y 319.595,Z 229.669,A -85,B 0,C 180,E1 -15137.931,E2 -15137.931} C_VEL
LIN {X 0,Y 319.546,Z 229.672,A -85,B 0,C 180,E1 -15141.956,E2 -15141.956} C_VEL
LIN {X 0,Y 319.537,Z 229.673,A -85,B 0,C 180,E1 -15146.097,E2 -15146.097} C_VEL
LIN {X 0,Y 319.509,Z 229.68,A -85,B 0,C 180,E1 -15148.942,E2 -15148.942} C_VEL
LIN {X 0,Y 319.504,Z 229.686,A -85,B 0,C 180,E1 -15151.865,E2 -15151.865} C_VEL
LIN {X 0,Y 319.566,Z 229.677,A -85,B 0,C 180,E1 -15155.543,E2 -15155.543} C_VEL
LIN {X 0,Y 319.55,Z 229.664,A -85,B 0,C 180,E1 -15159.67,E2 -15159.67} C_VEL
LIN {X 0,Y 319.512,Z 229.684,A -85,B 0,C 180,E1 -15163.461,E2 -15163.461} C_VEL
LIN {X 0,Y 319.545,Z 229.679,A -85,B 0,C 180,E1 -15167.017,E2 -15167.017} C_VEL
LIN {X 0,Y 319.51,Z 229.686,A -85,B 0,C 180,E1 -15170.367,E2 -15170.367} C_VEL
LIN {X 0,Y 319.575,Z 229.672,A -85,B 0,C 180,E1 -15174.458,E2 -15174.458} C_VEL
LIN {X 0,Y 319.591,Z 229.692,A -85,B 0,C 180,E1 -15174.6,E2 -15174.6} C_VEL
LIN {X 0,Y 322.44,Z 241.1,A -85,B 0,C 180,E1 -15178.218,E2 -15178.218} C_VEL
LIN {X 0,Y 325.013,Z 252.463,A -85,B 0,C 180,E1 -15181.594,E2 -15181.594} C_VEL
LIN {X 0,Y 325.709,Z 258.288,A -85,B 0,C 180,E1 -15183.202,E2 -15183.202} C_VEL
LIN {X 0,Y 325.662,Z 258.746,A -85,B 0,C 180,E1 -15183.318,E2 -15183.318} C_VEL
LIN {X 0,Y 331.173,Z 285.565,A -85,B 0,C 180,E1 -15184.536,E2 -15184.536} C_VEL
LIN {X 0,Y 333.956,Z 303.289,A -85,B 0,C 180,E1 -15185.228,E2 -15185.228} C_VEL
LIN {X 0,Y 332.225,Z 368.404,A -85,B 0,C 180,E1 -15186.673,E2 -15186.673} C_VEL
LIN {X 0,Y 331.207,Z 382.135,A -85,B 0,C 180,E1 -15187.216,E2 -15187.216} C_VEL
LIN {X 0,Y 329.941,Z 394.487,A -85,B 0,C 180,E1 -15187.949,E2 -15187.949} C_VEL
LIN {X 0,Y 328.445,Z 405.549,A -85,B 0,C 180,E1 -15188.833,E2 -15188.833} C_VEL
LIN {X 0,Y 326.618,Z 417.085,A -85,B 0,C 180,E1 -15190.026,E2 -15190.026} C_VEL
LIN {X 0,Y 324.926,Z 427.486,A -85,B 0,C 180,E1 -15191.395,E2 -15191.395} C_VEL
LIN {X 0,Y 323.114,Z 437.218,A -85,B 0,C 180,E1 -15192.989,E2 -15192.989} C_VEL
LIN {X 0,Y 321.615,Z 445.977,A -85,B 0,C 180,E1 -15194.797,E2 -15194.797} C_VEL
LIN {X 0,Y 320.269,Z 453.329,A -85,B 0,C 180,E1 -15196.678,E2 -15196.678} C_VEL
LIN {X 0,Y 319.153,Z 459.25,A -85,B 0,C 180,E1 -15198.568,E2 -15198.568} C_VEL
LIN {X 0,Y 318.494,Z 463.947,A -85,B 0,C 180,E1 -15200.472,E2 -15200.472} C_VEL
LIN {X 0,Y 318.064,Z 467.552,A -85,B 0,C 180,E1 -15202.38,E2 -15202.38} C_VEL
LIN {X 0,Y 317.842,Z 470.158,A -85,B 0,C 180,E1 -15204.282,E2 -15204.282} C_VEL
LIN {X 0,Y 317.842,Z 471.85,A -85,B 0,C 180,E1 -15206.194,E2 -15206.194} C_VEL
LIN {X 0,Y 317.867,Z 472.717,A -85,B 0,C 180,E1 -15208.731,E2 -15208.731} C_VEL
LIN {X 0,Y 317.951,Z 472.521,A -85,B 0,C 180,E1 -15209.998,E2 -15209.998} C_VEL
LIN {X 0,Y 317.911,Z 471.925,A -85,B 0,C 180,E1 -15211.264,E2 -15211.264} C_VEL
LIN {X 0,Y 317.849,Z 470.933,A -85,B 0,C 180,E1 -15212.532,E2 -15212.532} C_VEL
LIN {X 0,Y 317.898,Z 469.536,A -85,B 0,C 180,E1 -15213.8,E2 -15213.8} C_VEL
LIN {X 0,Y 317.904,Z 466.352,A -85,B 0,C 180,E1 -15215.829,E2 -15215.829} C_VEL
LIN {X 0,Y 318.055,Z 462.559,A -85,B 0,C 180,E1 -15217.616,E2 -15217.616} C_VEL
LIN {X 0,Y 318.458,Z 456.354,A -85,B 0,C 180,E1 -15219.845,E2 -15219.845} C_VEL
LIN {X 0,Y 319.018,Z 449.566,A -85,B 0,C 180,E1 -15221.754,E2 -15221.754} C_VEL
LIN {X 0,Y 319.948,Z 441.142,A -85,B 0,C 180,E1 -15223.655,E2 -15223.655} C_VEL
LIN {X 0,Y 320.852,Z 432.44,A -85,B 0,C 180,E1 -15225.235,E2 -15225.235} C_VEL
LIN {X 0,Y 322.061,Z 421.714,A -85,B 0,C 180,E1 -15226.802,E2 -15226.802} C_VEL
LIN {X 0,Y 323.167,Z 411.054,A -85,B 0,C 180,E1 -15228.049,E2 -15228.049} C_VEL
LIN {X 0,Y 324.397,Z 399.213,A -85,B 0,C 180,E1 -15229.124,E2 -15229.124} C_VEL
LIN {X 0,Y 325.398,Z 386.867,A -85,B 0,C 180,E1 -15229.965,E2 -15229.965} C_VEL
LIN {X 0,Y 326.209,Z 374.256,A -85,B 0,C 180,E1 -15230.571,E2 -15230.571} C_VEL
LIN {X 0,Y 326.669,Z 361.29,A -85,B 0,C 180,E1 -15230.953,E2 -15230.953} C_VEL
LIN {X 0,Y 327.581,Z 299.751,A -85,B 0,C 180,E1 -15232.299,E2 -15232.299} C_VEL
LIN {X 0,Y 322.306,Z 259.533,A -85,B 0,C 180,E1 -15233.557,E2 -15233.557} C_VEL
LIN {X 0,Y 323.356,Z 249.168,A -85,B 0,C 180,E1 -15236.069,E2 -15236.069} C_VEL
LIN {X 0,Y 322.15,Z 241.933,A -85,B 0,C 180,E1 -15237.967,E2 -15237.967} C_VEL
LIN {X 0,Y 319.646,Z 230.137,A -85,B 0,C 180,E1 -15241.185,E2 -15241.185} C_VEL
LIN {X 0,Y 319.552,Z 229.685,A -85,B 0,C 180,E1 -15241.349,E2 -15241.349} C_VEL
LIN {X 0,Y 319.542,Z 229.68,A -85,B 0,C 180,E1 -15244.872,E2 -15244.872} C_VEL
LIN {X 0,Y 319.552,Z 229.683,A -85,B 0,C 180,E1 -15248.004,E2 -15248.004} C_VEL
LIN {X 0,Y 319.503,Z 229.687,A -85,B 0,C 180,E1 -15251.592,E2 -15251.592} C_VEL
LIN {X 0,Y 319.533,Z 229.681,A -85,B 0,C 180,E1 -15255.265,E2 -15255.265} C_VEL
LIN {X 0,Y 319.551,Z 229.678,A -85,B 0,C 180,E1 -15258.715,E2 -15258.715} C_VEL
LIN {X 0,Y 319.55,Z 229.678,A -85,B 0,C 180,E1 -15262.339,E2 -15262.339} C_VEL
LIN {X 0,Y 319.526,Z 229.682,A -85,B 0,C 180,E1 -15265.119,E2 -15265.119} C_VEL
LIN {X 0,Y 319.534,Z 229.681,A -85,B 0,C 180,E1 -15269.055,E2 -15269.055} C_VEL
LIN {X 0,Y 319.57,Z 229.675,A -85,B 0,C 180,E1 -15272.495,E2 -15272.495} C_VEL
LIN {X 0,Y 319.585,Z 229.677,A -85,B 0,C 180,E1 -15275.302,E2 -15275.302} C_VEL
LIN {X 0,Y 319.608,Z 229.671,A -85,B 0,C 180,E1 -15278.049,E2 -15278.049} C_VEL
LIN {X 0,Y 319.651,Z 229.667,A -85,B 0,C 180,E1 -15280.959,E2 -15280.959} C_VEL
LIN {X 0,Y 319.688,Z 229.665,A -85,B 0,C 180,E1 -15285.275,E2 -15285.275} C_VEL
LIN {X 0,Y 319.714,Z 229.658,A -85,B 0,C 180,E1 -15289.872,E2 -15289.872} C_VEL
LIN {X 0,Y 319.886,Z 229.635,A -85,B 0,C 180,E1 -15292.425,E2 -15292.425} C_VEL
LIN {X 0,Y 319.705,Z 229.662,A -85,B 0,C 180,E1 -15294.956,E2 -15294.956} C_VEL
LIN {X 0,Y 319.944,Z 229.63,A -85,B 0,C 180,E1 -15297.482,E2 -15297.482} C_VEL
LIN {X 0,Y 320.083,Z 229.608,A -85,B 0,C 180,E1 -15300,E2 -15300} C_VEL
LIN {X 0,Y 319.939,Z 229.624,A -85,B 0,C 180,E1 -15302.518,E2 -15302.518} C_VEL
LIN {X 0,Y 319.868,Z 229.636,A -85,B 0,C 180,E1 -15306.686,E2 -15306.686} C_VEL
LIN {X 0,Y 319.708,Z 229.658,A -85,B 0,C 180,E1 -15310.129,E2 -15310.129} C_VEL
LIN {X 0,Y 319.687,Z 229.655,A -85,B 0,C 180,E1 -15313.994,E2 -15313.994} C_VEL
LIN {X 0,Y 319.578,Z 229.673,A -85,B 0,C 180,E1 -15317.932,E2 -15317.932} C_VEL
LIN {X 0,Y 319.525,Z 229.681,A -85,B 0,C 180,E1 -15321.958,E2 -15321.958} C_VEL
LIN {X 0,Y 319.581,Z 229.675,A -85,B 0,C 180,E1 -15326.093,E2 -15326.093} C_VEL
LIN {X 0,Y 319.553,Z 229.678,A -85,B 0,C 180,E1 -15328.938,E2 -15328.938} C_VEL
LIN {X 0,Y 319.497,Z 229.685,A -85,B 0,C 180,E1 -15331.866,E2 -15331.866} C_VEL
LIN {X 0,Y 319.547,Z 229.678,A -85,B 0,C 180,E1 -15335.547,E2 -15335.547} C_VEL
LIN {X 0,Y 319.552,Z 229.68,A -85,B 0,C 180,E1 -15338.011,E2 -15338.011} C_VEL
LIN {X 0,Y 319.569,Z 229.675,A -85,B 0,C 180,E1 -15341.616,E2 -15341.616} C_VEL
LIN {X 0,Y 319.504,Z 229.68,A -85,B 0,C 180,E1 -15345.269,E2 -15345.269} C_VEL
LIN {X 0,Y 319.506,Z 229.684,A -85,B 0,C 180,E1 -15348.716,E2 -15348.716} C_VEL
LIN {X 0,Y 319.535,Z 229.68,A -85,B 0,C 180,E1 -15352.355,E2 -15352.355} C_VEL
LIN {X 0,Y 319.543,Z 229.678,A -85,B 0,C 180,E1 -15355.128,E2 -15355.128} C_VEL
LIN {X 0,Y 319.552,Z 229.677,A -85,B 0,C 180,E1 -15359.064,E2 -15359.064} C_VEL
LIN {X 0,Y 319.594,Z 229.673,A -85,B 0,C 180,E1 -15362.502,E2 -15362.502} C_VEL
LIN {X 0,Y 319.594,Z 229.672,A -85,B 0,C 180,E1 -15365.308,E2 -15365.308} C_VEL
LIN {X 0,Y 319.575,Z 229.676,A -85,B 0,C 180,E1 -15369.403,E2 -15369.403} C_VEL
LIN {X 0,Y 319.653,Z 229.668,A -85,B 0,C 180,E1 -15373.396,E2 -15373.396} C_VEL
LIN {X 0,Y 319.768,Z 229.783,A -85,B 0,C 180,E1 -15376.621,E2 -15376.621} C_VEL
LIN {X 0,Y 320.263,Z 232.412,A -85,B 0,C 180,E1 -15377.398,E2 -15377.398} C_VEL
LIN {X 0,Y 327.078,Z 252.346,A -85,B 0,C 180,E1 -15378.306,E2 -15378.306} C_VEL
LIN {X 0,Y 328.422,Z 261.006,A -85,B 0,C 180,E1 -15378.586,E2 -15378.586} C_VEL
LIN {X 0,Y 326.73,Z 339.095,A -85,B 0,C 180,E1 -15380.29,E2 -15380.29} C_VEL
LIN {X 0,Y 326.093,Z 352.538,A -85,B 0,C 180,E1 -15380.818,E2 -15380.818} C_VEL
LIN {X 0,Y 325.442,Z 364.688,A -85,B 0,C 180,E1 -15381.543,E2 -15381.543} C_VEL
LIN {X 0,Y 324.686,Z 376.945,A -85,B 0,C 180,E1 -15382.541,E2 -15382.541} C_VEL
LIN {X 0,Y 323.435,Z 388.56,A -85,B 0,C 180,E1 -15383.766,E2 -15383.766} C_VEL
LIN {X 0,Y 322.34,Z 398.97,A -85,B 0,C 180,E1 -15385.156,E2 -15385.156} C_VEL
LIN {X 0,Y 321.346,Z 407.492,A -85,B 0,C 180,E1 -15386.555,E2 -15386.555} C_VEL
LIN {X 0,Y 320.537,Z 415.331,A -85,B 0,C 180,E1 -15388.118,E2 -15388.118} C_VEL
LIN {X 0,Y 319.554,Z 423.029,A -85,B 0,C 180,E1 -15390.002,E2 -15390.002} C_VEL
LIN {X 0,Y 318.968,Z 429.185,A -85,B 0,C 180,E1 -15391.896,E2 -15391.896} C_VEL
LIN {X 0,Y 318.472,Z 434.092,A -85,B 0,C 180,E1 -15393.798,E2 -15393.798} C_VEL
LIN {X 0,Y 318.201,Z 438.255,A -85,B 0,C 180,E1 -15395.931,E2 -15395.931} C_VEL
LIN {X 0,Y 317.992,Z 440.653,A -85,B 0,C 180,E1 -15397.622,E2 -15397.622} C_VEL
LIN {X 0,Y 317.847,Z 441.97,A -85,B 0,C 180,E1 -15398.906,E2 -15398.906} C_VEL
LIN {X 0,Y 317.776,Z 442.893,A -85,B 0,C 180,E1 -15400.192,E2 -15400.192} C_VEL
LIN {X 0,Y 317.812,Z 443.386,A -85,B 0,C 180,E1 -15401.481,E2 -15401.481} C_VEL
LIN {X 0,Y 317.955,Z 443.371,A -85,B 0,C 180,E1 -15403.451,E2 -15403.451} C_VEL
LIN {X 0,Y 318.173,Z 442.442,A -85,B 0,C 180,E1 -15405.372,E2 -15405.372} C_VEL
LIN {X 0,Y 318.399,Z 441.278,A -85,B 0,C 180,E1 -15406.676,E2 -15406.676} C_VEL
LIN {X 0,Y 319.002,Z 438.66,A -85,B 0,C 180,E1 -15408.675,E2 -15408.675} C_VEL
LIN {X 0,Y 319.73,Z 435.126,A -85,B 0,C 180,E1 -15410.592,E2 -15410.592} C_VEL
LIN {X 0,Y 320.713,Z 430.379,A -85,B 0,C 180,E1 -15412.537,E2 -15412.537} C_VEL
LIN {X 0,Y 321.954,Z 424.226,A -85,B 0,C 180,E1 -15414.504,E2 -15414.504} C_VEL
LIN {X 0,Y 323.527,Z 416.55,A -85,B 0,C 180,E1 -15416.444,E2 -15416.444} C_VEL
LIN {X 0,Y 325.025,Z 408.6,A -85,B 0,C 180,E1 -15418.061,E2 -15418.061} C_VEL
LIN {X 0,Y 326.669,Z 398.864,A -85,B 0,C 180,E1 -15419.658,E2 -15419.658} C_VEL
LIN {X 0,Y 328.477,Z 387.769,A -85,B 0,C 180,E1 -15421.099,E2 -15421.099} C_VEL
LIN {X 0,Y 329.907,Z 377.295,A -85,B 0,C 180,E1 -15422.179,E2 -15422.179} C_VEL
LIN {X 0,Y 331.047,Z 365.456,A -85,B 0,C 180,E1 -15423.137,E2 -15423.137} C_VEL
LIN {X 0,Y 332.177,Z 352.255,A -85,B 0,C 180,E1 -15423.902,E2 -15423.902} C_VEL
LIN {X 0,Y 332.841,Z 339.922,A -85,B 0,C 180,E1 -15424.382,E2 -15424.382} C_VEL
LIN {X 0,Y 334.932,Z 264.524,A -85,B 0,C 180,E1 -15426.03,E2 -15426.03} C_VEL
LIN {X 0,Y 327.761,Z 248.063,A -85,B 0,C 180,E1 -15427.143,E2 -15427.143} C_VEL
LIN {X 0,Y 325.658,Z 245.131,A -85,B 0,C 180,E1 -15427.434,E2 -15427.434} C_VEL
LIN {X 0,Y 320.926,Z 241.662,A -85,B 0,C 180,E1 -15428.026,E2 -15428.026} C_VEL
LIN {X 0,Y 316.17,Z 238.24,A -85,B 0,C 180,E1 -15428.642,E2 -15428.642} C_VEL
LIN {X 0,Y 314.024,Z 235.367,A -85,B 0,C 180,E1 -15428.962,E2 -15428.962} C_VEL
LIN {X 0,Y 313.277,Z 233.588,A -85,B 0,C 180,E1 -15429.136,E2 -15429.136} C_VEL
LIN {X 0,Y 312.49,Z 230.555,A -85,B 0,C 180,E1 -15430.231,E2 -15430.231} C_VEL
LIN {X 0,Y 312.526,Z 230.545,A -85,B 0,C 180,E1 -15433.977,E2 -15433.977} C_VEL
LIN {X 0,Y 312.542,Z 230.553,A -85,B 0,C 180,E1 -15437.904,E2 -15437.904} C_VEL
LIN {X 0,Y 312.534,Z 230.553,A -85,B 0,C 180,E1 -15441.907,E2 -15441.907} C_VEL
LIN {X 0,Y 312.495,Z 230.554,A -85,B 0,C 180,E1 -15445.788,E2 -15445.788} C_VEL
LIN {X 0,Y 312.511,Z 230.55,A -85,B 0,C 180,E1 -15448.852,E2 -15448.852} C_VEL
LIN {X 0,Y 312.561,Z 230.546,A -85,B 0,C 180,E1 -15451.823,E2 -15451.823} C_VEL
LIN {X 0,Y 312.57,Z 230.548,A -85,B 0,C 180,E1 -15454.709,E2 -15454.709} C_VEL
LIN {X 0,Y 312.508,Z 230.556,A -85,B 0,C 180,E1 -15458.91,E2 -15458.91} C_VEL
LIN {X 0,Y 312.576,Z 230.546,A -85,B 0,C 180,E1 -15461.652,E2 -15461.652} C_VEL
LIN {X 0,Y 312.667,Z 230.533,A -85,B 0,C 180,E1 -15465.685,E2 -15465.685} C_VEL
LIN {X 0,Y 312.67,Z 230.531,A -85,B 0,C 180,E1 -15469.641,E2 -15469.641} C_VEL
LIN {X 0,Y 312.826,Z 230.515,A -85,B 0,C 180,E1 -15472.253,E2 -15472.253} C_VEL
LIN {X 0,Y 312.879,Z 230.503,A -85,B 0,C 180,E1 -15473.551,E2 -15473.551} C_VEL
LIN {X 0,Y 312.911,Z 230.5,A -85,B 0,C 180,E1 -15477.425,E2 -15477.425} C_VEL
LIN {X 0,Y 313.045,Z 230.489,A -85,B 0,C 180,E1 -15480,E2 -15480} C_VEL
LIN {X 0,Y 312.909,Z 230.5,A -85,B 0,C 180,E1 -15482.575,E2 -15482.575} C_VEL
LIN {X 0,Y 312.826,Z 230.516,A -85,B 0,C 180,E1 -15486.45,E2 -15486.45} C_VEL
LIN {X 0,Y 312.666,Z 230.536,A -85,B 0,C 180,E1 -15490.359,E2 -15490.359} C_VEL
LIN {X 0,Y 312.65,Z 230.541,A -85,B 0,C 180,E1 -15494.864,E2 -15494.864} C_VEL
LIN {X 0,Y 312.53,Z 230.555,A -85,B 0,C 180,E1 -15499.192,E2 -15499.192} C_VEL
LIN {X 0,Y 312.501,Z 230.556,A -85,B 0,C 180,E1 -15502.776,E2 -15502.776} C_VEL
LIN {X 0,Y 312.471,Z 230.558,A -85,B 0,C 180,E1 -15506.733,E2 -15506.733} C_VEL
LIN {X 0,Y 312.451,Z 230.556,A -85,B 0,C 180,E1 -15509.66,E2 -15509.66} C_VEL
LIN {X 0,Y 312.507,Z 230.549,A -85,B 0,C 180,E1 -15513.689,E2 -15513.689} C_VEL
LIN {X 0,Y 312.503,Z 230.54,A -85,B 0,C 180,E1 -15517.388,E2 -15517.388} C_VEL
LIN {X 0,Y 312.48,Z 230.557,A -85,B 0,C 180,E1 -15520.711,E2 -15520.711} C_VEL
LIN {X 0,Y 312.443,Z 230.568,A -85,B 0,C 180,E1 -15524.211,E2 -15524.211} C_VEL
LIN {X 0,Y 312.448,Z 230.554,A -85,B 0,C 180,E1 -15527.926,E2 -15527.926} C_VEL
LIN {X 0,Y 312.471,Z 230.554,A -85,B 0,C 180,E1 -15531.926,E2 -15531.926} C_VEL
LIN {X 0,Y 312.539,Z 230.599,A -85,B 0,C 180,E1 -15533.928,E2 -15533.928} C_VEL
LIN {X 0,Y 315.154,Z 240.711,A -85,B 0,C 180,E1 -15537.264,E2 -15537.264} C_VEL
LIN {X 0,Y 317.799,Z 252.515,A -85,B 0,C 180,E1 -15540.888,E2 -15540.888} C_VEL
LIN {X 0,Y 318.864,Z 258.436,A -85,B 0,C 180,E1 -15542.598,E2 -15542.598} C_VEL
LIN {X 0,Y 321.03,Z 267.125,A -85,B 0,C 180,E1 -15543.054,E2 -15543.054} C_VEL
LIN {X 0,Y 326.041,Z 292.958,A -85,B 0,C 180,E1 -15544.219,E2 -15544.219} C_VEL
LIN {X 0,Y 327.689,Z 304.873,A -85,B 0,C 180,E1 -15544.675,E2 -15544.675} C_VEL
LIN {X 0,Y 325.915,Z 368.267,A -85,B 0,C 180,E1 -15546.109,E2 -15546.109} C_VEL
LIN {X 0,Y 324.858,Z 381.935,A -85,B 0,C 180,E1 -15546.661,E2 -15546.661} C_VEL
LIN {X 0,Y 323.538,Z 394.248,A -85,B 0,C 180,E1 -15547.405,E2 -15547.405} C_VEL
LIN {X 0,Y 321.874,Z 406.073,A -85,B 0,C 180,E1 -15548.379,E2 -15548.379} C_VEL
LIN {X 0,Y 319.971,Z 417.454,A -85,B 0,C 180,E1 -15549.593,E2 -15549.593} C_VEL
LIN {X 0,Y 318.215,Z 427.732,A -85,B 0,C 180,E1 -15550.988,E2 -15550.988} C_VEL
LIN {X 0,Y 316.326,Z 437.322,A -85,B 0,C 180,E1 -15552.612,E2 -15552.612} C_VEL
LIN {X 0,Y 314.737,Z 446.004,A -85,B 0,C 180,E1 -15554.456,E2 -15554.456} C_VEL
LIN {X 0,Y 313.335,Z 453.29,A -85,B 0,C 180,E1 -15556.377,E2 -15556.377} C_VEL
LIN {X 0,Y 312.157,Z 459.154,A -85,B 0,C 180,E1 -15558.308,E2 -15558.308} C_VEL
LIN {X 0,Y 311.45,Z 463.801,A -85,B 0,C 180,E1 -15560.255,E2 -15560.255} C_VEL
LIN {X 0,Y 311.007,Z 467.36,A -85,B 0,C 180,E1 -15562.206,E2 -15562.206} C_VEL
LIN {X 0,Y 310.739,Z 470.156,A -85,B 0,C 180,E1 -15564.356,E2 -15564.356} C_VEL
LIN {X 0,Y 310.749,Z 471.573,A -85,B 0,C 180,E1 -15566.107,E2 -15566.107} C_VEL
LIN {X 0,Y 310.734,Z 472.182,A -85,B 0,C 180,E1 -15567.405,E2 -15567.405} C_VEL
LIN {X 0,Y 310.774,Z 472.384,A -85,B 0,C 180,E1 -15568.702,E2 -15568.702} C_VEL
LIN {X 0,Y 310.86,Z 472.163,A -85,B 0,C 180,E1 -15569.998,E2 -15569.998} C_VEL
LIN {X 0,Y 310.815,Z 471.545,A -85,B 0,C 180,E1 -15571.293,E2 -15571.293} C_VEL
LIN {X 0,Y 310.768,Z 470.533,A -85,B 0,C 180,E1 -15572.59,E2 -15572.59} C_VEL
LIN {X 0,Y 310.804,Z 469.098,A -85,B 0,C 180,E1 -15573.887,E2 -15573.887} C_VEL
LIN {X 0,Y 310.805,Z 466.229,A -85,B 0,C 180,E1 -15575.765,E2 -15575.765} C_VEL
LIN {X 0,Y 310.995,Z 462.036,A -85,B 0,C 180,E1 -15577.79,E2 -15577.79} C_VEL
LIN {X 0,Y 311.411,Z 455.761,A -85,B 0,C 180,E1 -15580.07,E2 -15580.07} C_VEL
LIN {X 0,Y 312.031,Z 448.916,A -85,B 0,C 180,E1 -15582.021,E2 -15582.021} C_VEL
LIN {X 0,Y 312.863,Z 441.939,A -85,B 0,C 180,E1 -15583.639,E2 -15583.639} C_VEL
LIN {X 0,Y 313.788,Z 433.514,A -85,B 0,C 180,E1 -15585.254,E2 -15585.254} C_VEL
LIN {X 0,Y 314.973,Z 423.148,A -85,B 0,C 180,E1 -15586.858,E2 -15586.858} C_VEL
LIN {X 0,Y 316.092,Z 412.865,A -85,B 0,C 180,E1 -15588.132,E2 -15588.132} C_VEL
LIN {X 0,Y 317.28,Z 401.641,A -85,B 0,C 180,E1 -15589.233,E2 -15589.233} C_VEL
LIN {X 0,Y 318.387,Z 389.102,A -85,B 0,C 180,E1 -15590.171,E2 -15590.171} C_VEL
LIN {X 0,Y 319.262,Z 376.61,A -85,B 0,C 180,E1 -15590.829,E2 -15590.829} C_VEL
LIN {X 0,Y 319.833,Z 364.06,A -85,B 0,C 180,E1 -15591.253,E2 -15591.253} C_VEL
LIN {X 0,Y 320.855,Z 300.642,A -85,B 0,C 180,E1 -15592.675,E2 -15592.675} C_VEL
LIN {X 0,Y 315.456,Z 259.166,A -85,B 0,C 180,E1 -15594.015,E2 -15594.015} C_VEL
LIN {X 0,Y 316.379,Z 249.678,A -85,B 0,C 180,E1 -15596.372,E2 -15596.372} C_VEL
LIN {X 0,Y 314.191,Z 238.272,A -85,B 0,C 180,E1 -15599.473,E2 -15599.473} C_VEL
LIN {X 0,Y 312.515,Z 230.561,A -85,B 0,C 180,E1 -15601.687,E2 -15601.687} C_VEL
LIN {X 0,Y 312.513,Z 230.559,A -85,B 0,C 180,E1 -15605.775,E2 -15605.775} C_VEL
LIN {X 0,Y 312.486,Z 230.558,A -85,B 0,C 180,E1 -15609.023,E2 -15609.023} C_VEL
LIN {X 0,Y 312.47,Z 230.561,A -85,B 0,C 180,E1 -15612.426,E2 -15612.426} C_VEL
LIN {X 0,Y 312.504,Z 230.559,A -85,B 0,C 180,E1 -15616.017,E2 -15616.017} C_VEL
LIN {X 0,Y 312.501,Z 230.56,A -85,B 0,C 180,E1 -15619.865,E2 -15619.865} C_VEL
LIN {X 0,Y 312.509,Z 230.555,A -85,B 0,C 180,E1 -15622.612,E2 -15622.612} C_VEL
LIN {X 0,Y 312.486,Z 230.558,A -85,B 0,C 180,E1 -15626.308,E2 -15626.308} C_VEL
LIN {X 0,Y 312.509,Z 230.555,A -85,B 0,C 180,E1 -15630.346,E2 -15630.346} C_VEL
LIN {X 0,Y 312.567,Z 230.548,A -85,B 0,C 180,E1 -15634.061,E2 -15634.061} C_VEL
LIN {X 0,Y 312.588,Z 230.549,A -85,B 0,C 180,E1 -15637.529,E2 -15637.529} C_VEL
LIN {X 0,Y 312.597,Z 230.546,A -85,B 0,C 180,E1 -15641.654,E2 -15641.654} C_VEL
LIN {X 0,Y 312.65,Z 230.538,A -85,B 0,C 180,E1 -15645.684,E2 -15645.684} C_VEL
LIN {X 0,Y 312.659,Z 230.538,A -85,B 0,C 180,E1 -15649.64,E2 -15649.64} C_VEL
LIN {X 0,Y 312.825,Z 230.514,A -85,B 0,C 180,E1 -15652.253,E2 -15652.253} C_VEL
LIN {X 0,Y 312.675,Z 230.536,A -85,B 0,C 180,E1 -15654.842,E2 -15654.842} C_VEL
LIN {X 0,Y 312.944,Z 230.502,A -85,B 0,C 180,E1 -15658.713,E2 -15658.713} C_VEL
LIN {X 0,Y 312.943,Z 230.496,A -85,B 0,C 180,E1 -15661.287,E2 -15661.287} C_VEL
LIN {X 0,Y 312.665,Z 230.537,A -85,B 0,C 180,E1 -15665.159,E2 -15665.159} C_VEL
LIN {X 0,Y 312.831,Z 230.513,A -85,B 0,C 180,E1 -15666.668,E2 -15666.668} C_VEL
LIN {X 0,Y 312.654,Z 230.537,A -85,B 0,C 180,E1 -15670.36,E2 -15670.36} C_VEL
LIN {X 0,Y 312.625,Z 230.538,A -85,B 0,C 180,E1 -15674.866,E2 -15674.866} C_VEL
LIN {X 0,Y 312.506,Z 230.556,A -85,B 0,C 180,E1 -15679.194,E2 -15679.194} C_VEL
LIN {X 0,Y 312.486,Z 230.56,A -85,B 0,C 180,E1 -15682.782,E2 -15682.782} C_VEL
LIN {X 0,Y 312.559,Z 230.549,A -85,B 0,C 180,E1 -15685.936,E2 -15685.936} C_VEL
LIN {X 0,Y 312.51,Z 230.554,A -85,B 0,C 180,E1 -15689.654,E2 -15689.654} C_VEL
LIN {X 0,Y 312.487,Z 230.557,A -85,B 0,C 180,E1 -15693.693,E2 -15693.693} C_VEL
LIN {X 0,Y 312.509,Z 230.554,A -85,B 0,C 180,E1 -15697.388,E2 -15697.388} C_VEL
LIN {X 0,Y 312.498,Z 230.558,A -85,B 0,C 180,E1 -15700.708,E2 -15700.708} C_VEL
LIN {X 0,Y 312.499,Z 230.558,A -85,B 0,C 180,E1 -15704.202,E2 -15704.202} C_VEL
LIN {X 0,Y 312.464,Z 230.561,A -85,B 0,C 180,E1 -15707.923,E2 -15707.923} C_VEL
LIN {X 0,Y 312.479,Z 230.557,A -85,B 0,C 180,E1 -15710.976,E2 -15710.976} C_VEL
LIN {X 0,Y 312.514,Z 230.558,A -85,B 0,C 180,E1 -15714.225,E2 -15714.225} C_VEL
LIN {X 0,Y 312.489,Z 230.557,A -85,B 0,C 180,E1 -15717.339,E2 -15717.339} C_VEL
LIN {X 0,Y 312.532,Z 230.553,A -85,B 0,C 180,E1 -15721.284,E2 -15721.284} C_VEL
LIN {X 0,Y 312.575,Z 230.546,A -85,B 0,C 180,E1 -15724.715,E2 -15724.715} C_VEL
LIN {X 0,Y 312.557,Z 230.551,A -85,B 0,C 180,E1 -15727.532,E2 -15727.532} C_VEL
LIN {X 0,Y 312.562,Z 230.553,A -85,B 0,C 180,E1 -15731.656,E2 -15731.656} C_VEL
LIN {X 0,Y 312.69,Z 230.537,A -85,B 0,C 180,E1 -15736.022,E2 -15736.022} C_VEL
LIN {X 0,Y 312.707,Z 230.589,A -85,B 0,C 180,E1 -15736.271,E2 -15736.271} C_VEL
LIN {X 0,Y 313.131,Z 232.761,A -85,B 0,C 180,E1 -15736.931,E2 -15736.931} C_VEL
LIN {X 0,Y 320.578,Z 254.453,A -85,B 0,C 180,E1 -15737.949,E2 -15737.949} C_VEL
LIN {X 0,Y 321.687,Z 262.086,A -85,B 0,C 180,E1 -15738.198,E2 -15738.198} C_VEL
LIN {X 0,Y 319.957,Z 339.56,A -85,B 0,C 180,E1 -15739.923,E2 -15739.923} C_VEL
LIN {X 0,Y 319.3,Z 352.945,A -85,B 0,C 180,E1 -15740.462,E2 -15740.462} C_VEL
LIN {X 0,Y 318.625,Z 365.077,A -85,B 0,C 180,E1 -15741.201,E2 -15741.201} C_VEL
LIN {X 0,Y 317.964,Z 375.612,A -85,B 0,C 180,E1 -15742.063,E2 -15742.063} C_VEL
LIN {X 0,Y 316.862,Z 386.308,A -85,B 0,C 180,E1 -15743.156,E2 -15743.156} C_VEL
LIN {X 0,Y 315.791,Z 396.134,A -85,B 0,C 180,E1 -15744.415,E2 -15744.415} C_VEL
LIN {X 0,Y 314.74,Z 405.182,A -85,B 0,C 180,E1 -15745.841,E2 -15745.841} C_VEL
LIN {X 0,Y 313.783,Z 413.467,A -85,B 0,C 180,E1 -15747.435,E2 -15747.435} C_VEL
LIN {X 0,Y 312.795,Z 421.588,A -85,B 0,C 180,E1 -15749.359,E2 -15749.359} C_VEL
LIN {X 0,Y 312.022,Z 428.129,A -85,B 0,C 180,E1 -15751.293,E2 -15751.293} C_VEL
LIN {X 0,Y 311.568,Z 433.331,A -85,B 0,C 180,E1 -15753.235,E2 -15753.235} C_VEL
